FOR i := 1 TO 25 DO
	_Assertions.ThatBool(
		actual := _CollisionDictionary.ContainsKey(key := i),
		message := "Rebuild must preserve dictionary links"
	).IsTrue();
	_Assertions.ThatBool(
		actual := _CollisionSet.Contains(value := i),
		message := "Rebuild must preserve set links"
	).IsTrue();
END_FOR

_CollisionDictionary.Clear();
_CollisionSet.Clear();
_CollisionDictionary.SetCopy(key := _Scalar, value := _OtherScalar);
_CollisionSet.SetCopy(value := _Scalar);
_Assertions.ThatBool(
	actual := _CollisionDictionary.ContainsKey(key := _Scalar),
	message := "Dictionary comparer must survive Clear"
).IsTrue();
_Assertions.ThatBool(
	actual := _CollisionSet.Contains(value := _Scalar),
	message := "Set comparer must survive Clear"
).IsTrue();
END_METHOD

(*!
<summary>Uses matching hashes for cross-width integers, signed zero, NaN and empty descriptors.</summary>
<description>
Starts with independent fixture state. The harness clears persistent resources before publication, including
after an aborted call. Terminal OOM injection is reserved for an isolated test.
</description>
*)
METHOD PRIVATE hashEqualityRepresentations
_Dictionary.SetCopy(key := _SignedKey, value := _Scalar);
_Dictionary.SetCopy(key := _UnsignedKey, value := _OtherScalar);
_Set.SetCopy(value := _SignedKey);
_Set.SetCopy(value := _UnsignedKey);
_Assertions.ThatDInt(
	actual := _Dictionary.Length,
	message := "Equal integer widths must share a key"
).ToBe(expected := 1);
_Assertions.ThatDInt(
	actual := _Set.Length,
	message := "Equal integer widths must share an entry"
).ToBe(expected := 1);

_RealBits.Raw := TOF_Core.Reals.ZERO_BITS;
_Dictionary.SetCopy(key := _RealBits.Value, value := _Scalar);
_Set.SetCopy(value := _RealBits.Value);
_LongRealBits.Raw := NOT TOF_Core.LongReals.MAGNITUDE_MASK;
_Dictionary.SetCopy(key := _LongRealBits.Value, value := _OtherScalar);
_Set.SetCopy(value := _LongRealBits.Value);
_Assertions.ThatDInt(
	actual := _Dictionary.Length,
	message := "Signed floating zeros must share a key"
).ToBe(expected := 2);
_Assertions.ThatDInt(
	actual := _Set.Length,
	message := "Signed floating zeros must share an entry"
).ToBe(expected := 2);

_RealBits.Raw := TOF_Core.Reals.CANONICAL_NAN_BITS;
_LongRealBits.Raw := TOF_Core.LongReals.CANONICAL_NAN_BITS;
_Dictionary.SetCopy(key := _RealBits.Value, value := _Scalar);
_Dictionary.SetCopy(key := _LongRealBits.Value, value := _OtherScalar);
_Set.SetCopy(value := _RealBits.Value);
_Set.SetCopy(value := _LongRealBits.Value);
_Assertions.ThatDInt(
	actual := _Dictionary.Length,
	message := "Cross-width NaNs must share a key"
).ToBe(expected := 3);
_Assertions.ThatDInt(
	actual := _Set.Length,
	message := "Cross-width NaNs must share an entry"
).ToBe(expected := 3);

_Query.Reset();
_Dictionary.SetGeneric(key := _Query, value := _Query);
_Set.SetGeneric(value := _Query);
_Assertions.ThatBool(
	actual := _Dictionary.ContainsGenericKey(key := _Query),
	message := "Empty key must be searchable"
).IsTrue();
_Assertions.ThatBool(
	actual := _Set.ContainsGeneric(value := _Query),
	message := "Empty entry must be searchable"
).IsTrue();
_Assertions.ThatDInt(
	actual := _Dictionary.Length,
	message := "Empty must remain distinct from nonempty values"
).ToBe(expected := 4);
_Assertions.ThatDInt(
	actual := _Set.Length,
	message := "Empty must remain distinct from nonempty values"
).ToBe(expected := 4);
END_METHOD

(*!
<summary>Disposes shared key/value allocations once and retains same-allocation set ownership.</summary>
<description>
Starts with independent fixture state. The harness clears persistent resources before publication, including
after an aborted call. Terminal OOM injection is reserved for an isolated test.
</description>
*)
METHOD PRIVATE hashOwnershipAliases
VAR
	borrowedValue : TOF_Core.GENERIC_VALUE;
	pair : TOF_Core.GENERIC_KEY_VALUE_PAIR;
END_VAR
prepareOwnedValue();
borrowedValue := TOF_Core.GenericValueFactory.FromParts(
	genericTypeClass := _OwnedValue.TypeClass,
	address := _OwnedValue.Address,
	size := _OwnedValue.Size,
	memoryManagementBehavior := TOF_Core.GENERIC_MEMORY_MANAGEMENT_BEHAVIOR.STORE_ORIGINAL_REFERENCE_AND_NOT_OWNS_MEMORY
);
_Dictionary.SetGeneric(key := _OwnedValue, value := _OwnedValue);
_OwnedValue.Reset();
pair := _Dictionary.GetKeyValuePairByIndex(index := 0);
_Assertions.ThatBool(
	actual := pair.Key.IsMemoryOwner,
	message := "Shared pair ownership must belong to key"
).IsTrue();
_Assertions.ThatBool(
	actual := pair.Value.IsMemoryOwner,
	message := "Shared pair value must remain borrowed"
).IsFalse();
_Dictionary.SetGeneric(key := borrowedValue, value := borrowedValue);
_Assertions.ThatUDInt(
	actual := _CloneExitCount,
	message := "Retained pair storage must stay alive"
).ToBe(expected := 0);
_Dictionary.Clear();
_Assertions.ThatUDInt(
	actual := _CloneExitCount,
	message := "Shared pair must be destroyed once"
).ToBe(expected := 1);

prepareOwnedValue();
borrowedValue := TOF_Core.GenericValueFactory.FromParts(
	genericTypeClass := _OwnedValue.TypeClass,
	address := _OwnedValue.Address,
	size := _OwnedValue.Size,
	memoryManagementBehavior := TOF_Core.GENERIC_MEMORY_MANAGEMENT_BEHAVIOR.STORE_ORIGINAL_REFERENCE_AND_NOT_OWNS_MEMORY
);
_Set.SetGeneric(value := _OwnedValue);
_OwnedValue.Reset();
_Set.SetGeneric(value := borrowedValue);
_Assertions.ThatBool(
	actual := _Set.GetByIndex(index := 0).IsMemoryOwner,
	message := "Set replacement must preserve owner"
).IsTrue();
_Set.Clear();
_Assertions.ThatUDInt(
	actual := _CloneExitCount,
	message := "Retained set storage must be destroyed once"
).ToBe(expected := 2);
END_METHOD

(*!
<summary>Preserves ownership when replacing a stored value with its borrowed same-allocation alias.</summary>
<description>
Starts with independent fixture state. The harness clears persistent resources before publication, including
after an aborted call. Terminal OOM injection is reserved for an isolated test.
</description>
*)
METHOD PRIVATE listOwnershipReplacement
VAR
	borrowedValue : TOF_Core.GENERIC_VALUE;
END_VAR
prepareOwnedValue();
_List.AppendGeneric(value := _OwnedValue);
_OwnedValue.Reset();
borrowedValue := TOF_Core.GenericValueFactory.FromParts(
	genericTypeClass := _List.Get(index := 0).TypeClass,
	address := _List.Get(index := 0).Address,
	size := _List.Get(index := 0).Size,
	memoryManagementBehavior := TOF_Core.GENERIC_MEMORY_MANAGEMENT_BEHAVIOR.STORE_ORIGINAL_REFERENCE_AND_NOT_OWNS_MEMORY
);
_List.SetGeneric(index := 0, value := borrowedValue);
_Assertions.ThatBool(
	actual := _List.Get(index := 0).IsMemoryOwner,
	message := "Borrowed replacement must preserve owner"
).IsTrue();
_Assertions.ThatUDInt(
	actual := _CloneExitCount,
	message := "Same allocation must remain alive"
).ToBe(expected := 0);
_List.Clear();
_Assertions.ThatUDInt(
	actual := _CloneExitCount,
	message := "Retained allocation must be destroyed once"
).ToBe(expected := 1);
END_METHOD

(*!
<summary>Applies skip and maxRemoved and preserves completed removals after a predicate failure.</summary>
<description>
Starts with independent fixture state. The harness clears persistent resources before publication, including
after an aborted call. Terminal OOM injection is reserved for an isolated test.
</description>
*)
METHOD PRIVATE listRemovalLimits
VAR
	i : DINT;
	removedCount : DINT;
	rejected : BOOL;
	exceptionCode : __SYSTEM.ExceptionCode;
END_VAR
FOR i := 1 TO 5 DO
	_List.AppendCopy(value := i);
END_FOR

_Predicate.ResetCount();
_List.RemoveMatched(predicate := _Predicate, skip := 1, maxRemoved := 2, removedCount => removedCount);
_Assertions.ThatDInt(
	actual := removedCount,
	message := "Removal must obey the positive limit"
).ToBe(expected := 2);
_Assertions.ThatUDInt(
	actual := _Predicate.CallCount,
	message := "Limit must stop further callbacks"
).ToBe(expected := 3);
_Assertions.ThatDInt(
	actual := _List.Length,
	message := "Two matches must be removed"
).ToBe(expected := 3);
_Assertions.ThatDInt(
	actual := _List.Get(index := 2).AsDInt(),
	message := "Skipped last match must remain"
).ToBe(expected := 5);
_Predicate.ResetCount();
_List.RemoveMatched(predicate := _Predicate, maxRemoved := 0, removedCount => removedCount);
_Assertions.ThatUDInt(
	actual := _Predicate.CallCount,
	message := "Zero limit must not invoke predicate"
).ToBe(expected := 0);
_Assertions.ThatDInt(
	actual := removedCount,
	message := "Zero limit must report no removals"
).ToBe(expected := 0);

_List.Clear();

FOR i := 1 TO 5 DO
	_List.AppendCopy(value := i);
END_FOR

_Predicate.ResetCount();
_Predicate.ThrowOnCall := 2;

__TRY
	_List.RemoveMatched(predicate := _Predicate, removedCount => removedCount);
__CATCH(exceptionCode)
	rejected := TRUE;
	assertOriginalFailure(exceptionCode := exceptionCode, expectedMessage := "Collection predicate rejected");
__ENDTRY

_Assertions.ThatBool(
	actual := rejected,
	message := "Predicate failure must propagate"
).IsTrue();
_Assertions.ThatDInt(
	actual := _List.Length,
	message := "Completed removal must not roll back"
).ToBe(expected := 4);
_Assertions.ThatDInt(
	actual := _List.Get(index := 3).AsDInt(),
	message := "Remaining order must be valid"
).ToBe(expected := 4);
END_METHOD

(*!
<summary>Diagnoses null constructor sources outside FB_init for all six cursors and concrete current views.</summary>
<description>
All six cursors are constructed with null sources without throwing during FB_init. MoveNext, generic
Current and concrete current views must report configuration failure in the current cyclic task. Reset
remains a local cursor operation that does not access the missing source.
</description>
*)
METHOD PRIVATE missingCursorSources
VAR
	i : DINT;
	rejected : BOOL;
	exceptionCode : __SYSTEM.ExceptionCode;
	caughtException : TOF_Core.IException;
	missingException : TOF_Core.IDataMemberNotSpecifiedException;
	currentValue : TOF_Core.GENERIC_VALUE;
	currentByte : BYTE;
	currentPair : TOF_Core.GENERIC_KEY_VALUE_PAIR;
END_VAR
_NullCursors[0] := _NullByteCursor;
_NullCursors[1] := _NullListCursor;
_NullCursors[2] := _NullQueueCursor;
_NullCursors[3] := _NullStackCursor;
_NullCursors[4] := _NullDictionaryCursor;
_NullCursors[5] := _NullSetCursor;

FOR i := 0 TO 5 DO
	rejected := FALSE;

	__TRY
		_NullCursors[i].MoveNext();
	__CATCH(exceptionCode)
		rejected := TRUE;
		caughtException := TOF_Core.ExceptionManager.GetLastException(
			exceptionCode := exceptionCode,
			catchPointNamespaceName := NamespaceName,
			catchPointPOUName := __POUNAME(),
			catchPointPosition := __POSITION()
		);
		_Assertions.ThatBool(
			actual := __QUERYINTERFACE(caughtException, missingException),
			message := "Missing cursor source must report DataMemberNotSpecifiedException"
		).IsTrue();
	__ENDTRY

	_Assertions.ThatBool(
		actual := rejected,
		message := "MoveNext must reject a missing source"
	).IsTrue();
	rejected := FALSE;

	__TRY
		currentValue := _NullCursors[i].Current;
	__CATCH(exceptionCode)
		rejected := TRUE;
		caughtException := TOF_Core.ExceptionManager.GetLastException(
			exceptionCode := exceptionCode,
			catchPointNamespaceName := NamespaceName,
			catchPointPOUName := __POUNAME(),
			catchPointPosition := __POSITION()
		);
		_Assertions.ThatBool(
			actual := __QUERYINTERFACE(caughtException, missingException),
			message := "Missing cursor source must report DataMemberNotSpecifiedException"
		).IsTrue();
	__ENDTRY

	_Assertions.ThatBool(
		actual := rejected,
		message := "Current must reject a missing source"
	).IsTrue();
	_NullCursors[i].Reset();
END_FOR

rejected := FALSE;

__TRY
	currentByte := _NullByteCursor.CurrentByte;
__CATCH(exceptionCode)
	rejected := TRUE;
	caughtException := TOF_Core.ExceptionManager.GetLastException(
		exceptionCode := exceptionCode,
		catchPointNamespaceName := NamespaceName,
		catchPointPOUName := __POUNAME(),
		catchPointPosition := __POSITION()
	);
	_Assertions.ThatBool(
		actual := __QUERYINTERFACE(caughtException, missingException),
		message := "Missing cursor source must report DataMemberNotSpecifiedException"
	).IsTrue();
__ENDTRY

_Assertions.ThatBool(
	actual := rejected,
	message := "Concrete CurrentByte must reject a missing source"
).IsTrue();
rejected := FALSE;

__TRY
	currentPair := _NullDictionaryCursor.CurrentKeyValuePair;
__CATCH(exceptionCode)
	rejected := TRUE;
	caughtException := TOF_Core.ExceptionManager.GetLastException(
		exceptionCode := exceptionCode,
		catchPointNamespaceName := NamespaceName,
		catchPointPOUName := __POUNAME(),
		catchPointPosition := __POSITION()
	);
	_Assertions.ThatBool(
		actual := __QUERYINTERFACE(caughtException, missingException),
		message := "Missing cursor source must report DataMemberNotSpecifiedException"
	).IsTrue();
__ENDTRY

_Assertions.ThatBool(
	actual := rejected,
	message := "Concrete CurrentKeyValuePair must reject a missing source"
).IsTrue();
END_METHOD

(*!
<summary>Retains one clone as a fixture-owned descriptor until acceptance or cleanup.</summary>
*)
METHOD PRIVATE prepareOwnedValue
_OwnedObject := _CloneSource.Clone();
_OwnedValue := TOF_Core.GenericValueFactory.FromParts(
	genericTypeClass := TOF_Core.GENERIC_TYPE_CLASS.OBJECT,
	address := _OwnedObject.SelfAddress,
	size := _OwnedObject.SelfSize,
	memoryManagementBehavior := TOF_Core.GENERIC_MEMORY_MANAGEMENT_BEHAVIOR.STORE_ORIGINAL_REFERENCE_AND_OWNS_MEMORY
);
_OwnedObject := 0;
END_METHOD

(*!
<summary>Prepares persistent resources and raises before the caller can release them.</summary>
*)
METHOD PRIVATE prepareResourcesThenReject
_Enumerator := _List.CreateEnumerator();
prepareOwnedValue();
TOF_Core.Exceptions.ThrowStandard(
	sourceNamespaceName := NamespaceName,
	sourceClassName := ClassName,
	sourcePOUName := __POUNAME(),
	sourcePosition := __POSITION(),
	message := "Collection fixture rejected"
);
END_METHOD

(*!
<summary>Releases owned queries and retains callback diagnostics across cleanup context changes.</summary>
<description>
Starts with independent fixture state. The harness clears persistent resources before publication, including
after an aborted call. Terminal OOM injection is reserved for an isolated test.
</description>
*)
METHOD PRIVATE queryFailureCleanup
VAR
	rejected : BOOL;
	exceptionCode : __SYSTEM.ExceptionCode;
END_VAR
_BorrowedSource := TOF_Core.GenericValueFactory.FromParts(
	genericTypeClass := TOF_Core.GENERIC_TYPE_CLASS.OBJECT,
	address := _CloneSource.SelfAddress,
	size := _CloneSource.SelfSize,
	memoryManagementBehavior := TOF_Core.GENERIC_MEMORY_MANAGEMENT_BEHAVIOR.STORE_ORIGINAL_REFERENCE_AND_NOT_OWNS_MEMORY
);
_List.AppendGeneric(value := _BorrowedSource);
_Queue.EnqueueGeneric(value := _BorrowedSource);
_Stack.PushGeneric(value := _BorrowedSource);
_CollisionDictionary.SetCopy(key := _Scalar, value := _Scalar);
_CollisionSet.SetCopy(value := _Scalar);
_CloneSource.ThrowOnEquality := TRUE;
_Equality.ThrowOnEquality := TRUE;

prepareOwnedValue();
_Query := _OwnedValue;
_OwnedValue.Reset();

rejected := FALSE;
_CloneExitCount := TOF_Core.UnsignedInt32.ZERO;

__TRY
	_List.ContainsGeneric(value := _Query, releaseValue := TRUE);
	_Query.Reset();
__CATCH(exceptionCode)
	_Query.Reset();
	rejected := TRUE;
	assertOriginalFailure(exceptionCode := exceptionCode, expectedMessage := "Collection object equality rejected");
__ENDTRY

_Assertions.ThatBool(
	actual := rejected,
	message := "Failure must propagate"
).IsTrue();
_Assertions.ThatUDInt(
	actual := _CloneExitCount,
	message := "Owned temporary must be released exactly once"
).ToBe(expected := 1);

prepareOwnedValue();
_Query := _OwnedValue;
_OwnedValue.Reset();

rejected := FALSE;
_CloneExitCount := TOF_Core.UnsignedInt32.ZERO;

__TRY
	_Queue.ContainsGeneric(value := _Query, releaseValue := TRUE);
	_Query.Reset();
__CATCH(exceptionCode)
	_Query.Reset();
	rejected := TRUE;
	assertOriginalFailure(exceptionCode := exceptionCode, expectedMessage := "Collection object equality rejected");
__ENDTRY

_Assertions.ThatBool(
	actual := rejected,
	message := "Failure must propagate"
).IsTrue();
_Assertions.ThatUDInt(
	actual := _CloneExitCount,
	message := "Owned temporary must be released exactly once"
).ToBe(expected := 1);

prepareOwnedValue();
_Query := _OwnedValue;
_OwnedValue.Reset();

rejected := FALSE;
_CloneExitCount := TOF_Core.UnsignedInt32.ZERO;

__TRY
	_Stack.ContainsGeneric(value := _Query, releaseValue := TRUE);
	_Query.Reset();
__CATCH(exceptionCode)
	_Query.Reset();
	rejected := TRUE;
	assertOriginalFailure(exceptionCode := exceptionCode, expectedMessage := "Collection object equality rejected");
__ENDTRY

_Assertions.ThatBool(
	actual := rejected,
	message := "Failure must propagate"
).IsTrue();
_Assertions.ThatUDInt(
	actual := _CloneExitCount,
	message := "Owned temporary must be released exactly once"
).ToBe(expected := 1);

prepareOwnedValue();
_Query := _OwnedValue;
_OwnedValue.Reset();

rejected := FALSE;
_CloneExitCount := TOF_Core.UnsignedInt32.ZERO;

__TRY
	_CollisionDictionary.ContainsGenericKey(key := _Query, releaseKey := TRUE);
	_Query.Reset();
__CATCH(exceptionCode)
	_Query.Reset();
	rejected := TRUE;
	assertOriginalFailure(exceptionCode := exceptionCode, expectedMessage := "Collection equality rejected");
__ENDTRY

_Assertions.ThatBool(
	actual := rejected,
	message := "Failure must propagate"
).IsTrue();
_Assertions.ThatUDInt(
	actual := _CloneExitCount,
	message := "Owned temporary must be released exactly once"
).ToBe(expected := 1);

prepareOwnedValue();
_Query := _OwnedValue;
_OwnedValue.Reset();

rejected := FALSE;
_CloneExitCount := TOF_Core.UnsignedInt32.ZERO;

__TRY
	_CollisionDictionary.GetGenericKeyPosition(key := _Query, releaseKey := TRUE);
	_Query.Reset();
__CATCH(exceptionCode)
	_Query.Reset();
	rejected := TRUE;
	assertOriginalFailure(exceptionCode := exceptionCode, expectedMessage := "Collection equality rejected");
__ENDTRY

_Assertions.ThatBool(
	actual := rejected,
	message := "Failure must propagate"
).IsTrue();
_Assertions.ThatUDInt(
	actual := _CloneExitCount,
	message := "Owned temporary must be released exactly once"
).ToBe(expected := 1);

prepareOwnedValue();
_Query := _OwnedValue;
_OwnedValue.Reset();

rejected := FALSE;
_CloneExitCount := TOF_Core.UnsignedInt32.ZERO;

__TRY
	_CollisionSet.ContainsGeneric(value := _Query, releaseValue := TRUE);
	_Query.Reset();
__CATCH(exceptionCode)
	_Query.Reset();
	rejected := TRUE;
	assertOriginalFailure(exceptionCode := exceptionCode, expectedMessage := "Collection equality rejected");
__ENDTRY

_Assertions.ThatBool(
	actual := rejected,
	message := "Failure must propagate"
).IsTrue();
_Assertions.ThatUDInt(
	actual := _CloneExitCount,
	message := "Owned temporary must be released exactly once"
).ToBe(expected := 1);

prepareOwnedValue();
_Query := _OwnedValue;
_OwnedValue.Reset();

rejected := FALSE;
_CloneExitCount := TOF_Core.UnsignedInt32.ZERO;

__TRY
	_CollisionSet.GetGenericValuePosition(value := _Query, releaseValue := TRUE);
	_Query.Reset();
__CATCH(exceptionCode)
	_Query.Reset();
	rejected := TRUE;
	assertOriginalFailure(exceptionCode := exceptionCode, expectedMessage := "Collection equality rejected");
__ENDTRY

_Assertions.ThatBool(
	actual := rejected,
	message := "Failure must propagate"
).IsTrue();
_Assertions.ThatUDInt(
	actual := _CloneExitCount,
	message := "Owned temporary must be released exactly once"
).ToBe(expected := 1);

_Assertions.ThatDInt(
	actual := _List.Length,
	message := "Failed query must not remove list entries"
).ToBe(expected := 1);
_Assertions.ThatDInt(
	actual := _CollisionDictionary.Length,
	message := "Failed query must not mutate keys"
).ToBe(expected := 1);
_Assertions.ThatDInt(
	actual := _CollisionSet.Length,
	message := "Failed query must not mutate values"
).ToBe(expected := 1);
END_METHOD

(*!
<summary>Invokes the validator once per enqueue and rejects before growth or adoption.</summary>
<description>
Starts with independent fixture state. The harness clears persistent resources before publication, including
after an aborted call. Terminal OOM injection is reserved for an isolated test.
</description>
*)
METHOD PRIVATE queueValidationAndGrowth
VAR
	i : DINT;
	rejected : BOOL;
	exceptionCode : __SYSTEM.ExceptionCode;
END_VAR
_Queue.DefaultDynamicAllocationElementCount := 2;
_Validator.ResetCount();

FOR i := 1 TO 6 DO
	_Queue.EnqueueCopy(value := i);
END_FOR

_Assertions.ThatUDInt(
	actual := _Validator.CallCount,
	message := "Enqueue must validate exactly once"
).ToBe(expected := 6);
_Assertions.ThatDInt(
	actual := _Queue.Capacity,
	message := "Queue must grow several times"
).ToBe(expected := 6);
_Validator.Reject := TRUE;
prepareOwnedValue();

__TRY
	_Queue.EnqueueGeneric(value := _OwnedValue);
__CATCH(exceptionCode)
	rejected := TRUE;
	assertOriginalFailure(exceptionCode := exceptionCode, expectedMessage := "Collection validation rejected");
__ENDTRY

_Assertions.ThatBool(
	actual := rejected,
	message := "Configured validator must reject"
).IsTrue();
_Assertions.ThatDInt(
	actual := _Queue.Capacity,
	message := "Rejected enqueue must not grow"
).ToBe(expected := 6);
_Assertions.ThatDInt(
	actual := _Queue.Length,
	message := "Rejected enqueue must not insert"
).ToBe(expected := 6);
_Assertions.ThatUDInt(
	actual := _CloneExitCount,
	message := "Rejected owner must remain caller-owned"
).ToBe(expected := 0);
_OwnedValue.Release();
_Assertions.ThatUDInt(
	actual := _CloneExitCount,
	message := "Caller must retain disposal rights"
).ToBe(expected := 1);
_Validator.Reject := FALSE;

FOR i := 1 TO 6 DO
	_Assertions.ThatDInt(
		actual := _Queue.Peek().AsDInt(),
		message := "Growth must preserve FIFO order"
	).ToBe(expected := i);
	_Queue.RemoveFirst();
END_FOR
END_METHOD

(*!
<summary>Releases persistent cursor ownership without deleting source collections.</summary>
<description>
Clears interface aliases before best-effort disposal. Latches failed disposal or duplicate ownership.
</description>
*)
METHOD PRIVATE releaseCursors
VAR
	ownedCursor : TOF_Core.IObject;
END_VAR
IF _Enumerator <> 0 AND_THEN _Enumerator = _SecondEnumerator THEN
	_SecondEnumerator := 0;
	_ReleaseFailed := TRUE;
END_IF

IF _Enumerator <> 0 THEN
	ownedCursor := _Enumerator;
	_Enumerator := 0;

	IF NOT TOF_Core.Memory.TryReleaseDynamicObject(instance := ownedCursor) THEN
		_ReleaseFailed := TRUE;
	END_IF
END_IF

IF _SecondEnumerator <> 0 THEN
	ownedCursor := _SecondEnumerator;
	_SecondEnumerator := 0;

	IF NOT TOF_Core.Memory.TryReleaseDynamicObject(instance := ownedCursor) THEN
		_ReleaseFailed := TRUE;
	END_IF
END_IF
END_METHOD

(*!
<summary>Releases the prepared dictionary key if the second object clone rejects.</summary>
<description>
Starts with independent fixture state. The harness clears persistent resources before publication, including
after an aborted call. Terminal OOM injection is reserved for an isolated test.
</description>
*)
METHOD PRIVATE secondCopyFailureCleanup
VAR
	rejected : BOOL;
	exceptionCode : __SYSTEM.ExceptionCode;
END_VAR
_FailingCloneSource.ThrowOnClone := TRUE;

rejected := FALSE;
_CloneExitCount := TOF_Core.UnsignedInt32.ZERO;

__TRY
	_Dictionary.SetCopy(
		key := _CloneSource,
		value := _FailingCloneSource,
		keyIsObject := TRUE,
		valueIsObject := TRUE
	);
__CATCH(exceptionCode)
	rejected := TRUE;
	assertOriginalFailure(exceptionCode := exceptionCode, expectedMessage := "Collection clone rejected");
__ENDTRY

_Assertions.ThatBool(
	actual := rejected,
	message := "Failure must propagate"
).IsTrue();
_Assertions.ThatUDInt(
	actual := _CloneExitCount,
	message := "Owned temporary must be released exactly once"
).ToBe(expected := 1);

_Assertions.ThatBool(
	actual := _Dictionary.Empty,
	message := "Second clone failure must not insert a pair"
).IsTrue();
END_METHOD

(*!
<summary>Retains every owned descriptor after comparer failures in both sorting branches.</summary>
<description>
Starts with independent fixture state. The harness clears persistent resources before publication, including
after an aborted call. Terminal OOM injection is reserved for an isolated test.
</description>
*)
METHOD PRIVATE sortFailurePreservesEntries
VAR
	i : DINT;
	count : DINT;
	rejected : BOOL;
	exceptionCode : __SYSTEM.ExceptionCode;
END_VAR
FOR count := 16 TO 17 DO
	_List.Clear();

	FOR i := count TO 1 BY -1 DO
		_List.AppendCopy(value := i);
	END_FOR

	_Comparer.ResetCount();
	_Comparer.ThrowOnCall := 3;
	rejected := FALSE;

	__TRY
		_List.Sort(comparer := _Comparer);
	__CATCH(exceptionCode)
		rejected := TRUE;
		assertOriginalFailure(exceptionCode := exceptionCode, expectedMessage := "Collection comparer rejected");
	__ENDTRY

	_Assertions.ThatBool(
		actual := rejected,
		message := "Comparer failure must propagate"
	).IsTrue();
	_Assertions.ThatDInt(
		actual := _List.Length,
		message := "Failed sort must preserve Length"
	).ToBe(expected := count);
	_Comparer.ThrowOnCall := 0;
	_List.Sort(comparer := _Comparer);

	FOR i := 0 TO count - 1 DO
		_Assertions.ThatDInt(
			actual := _List.Get(index := i).AsDInt(),
			message := "Failed sorting must neither lose nor duplicate entries"
		).ToBe(expected := i + 1);
		_Assertions.ThatBool(
			actual := _List.Get(index := i).IsMemoryOwner,
			message := "Sorting must preserve ownership"
		).IsTrue();
	END_FOR
END_FOR
END_METHOD

(*!
<summary>Retains static-full diagnostics and disposes prepared copies before adoption.</summary>
<description>
Starts with independent fixture state. The harness clears persistent resources before publication, including
after an aborted call. Terminal OOM injection is reserved for an isolated test.
</description>
*)
METHOD PRIVATE staticFullCopyCleanup
VAR
	rejected : BOOL;
	exceptionCode : __SYSTEM.ExceptionCode;
	caughtException : TOF_Core.IException;
	fullException : TOF_Core.IStaticCollectionFullException;
END_VAR
_FullList.AppendCopy(value := _Scalar);
_FullQueue.EnqueueCopy(value := _Scalar);
_FullStack.PushCopy(value := _Scalar);
_FullDictionary.SetCopy(key := _Scalar, value := _Scalar);
_FullSet.SetCopy(value := _Scalar);

rejected := FALSE;
_CloneExitCount := TOF_Core.UnsignedInt32.ZERO;

__TRY
	_FullList.AppendCopy(value := _CloneSource, isObject := TRUE);
__CATCH(exceptionCode)
	rejected := TRUE;
	caughtException := TOF_Core.ExceptionManager.GetLastException(
		exceptionCode := exceptionCode,
		catchPointNamespaceName := NamespaceName,
		catchPointPOUName := __POUNAME(),
		catchPointPosition := __POSITION()
	);
	_Assertions.ThatBool(
		actual := __QUERYINTERFACE(caughtException, fullException),
		message := "Static-full diagnostic must survive clone disposal"
	).IsTrue();
__ENDTRY

_Assertions.ThatBool(
	actual := rejected,
	message := "Static full must reject Copy"
).IsTrue();
_Assertions.ThatUDInt(
	actual := _CloneExitCount,
	message := "Rejected copy must be released once"
).ToBe(expected := 1);

rejected := FALSE;
_CloneExitCount := TOF_Core.UnsignedInt32.ZERO;

__TRY
	_FullList.InsertCopy(index := 0, value := _CloneSource, isObject := TRUE);
__CATCH(exceptionCode)
	rejected := TRUE;
	caughtException := TOF_Core.ExceptionManager.GetLastException(
		exceptionCode := exceptionCode,
		catchPointNamespaceName := NamespaceName,
		catchPointPOUName := __POUNAME(),
		catchPointPosition := __POSITION()
	);
	_Assertions.ThatBool(
		actual := __QUERYINTERFACE(caughtException, fullException),
		message := "Static-full diagnostic must survive clone disposal"
	).IsTrue();
__ENDTRY

_Assertions.ThatBool(
	actual := rejected,
	message := "Static full must reject Copy"
).IsTrue();
_Assertions.ThatUDInt(
	actual := _CloneExitCount,
	message := "Rejected copy must be released once"
).ToBe(expected := 1);

rejected := FALSE;
_CloneExitCount := TOF_Core.UnsignedInt32.ZERO;

__TRY
	_FullQueue.EnqueueCopy(value := _CloneSource, isObject := TRUE);
__CATCH(exceptionCode)
	rejected := TRUE;
	caughtException := TOF_Core.ExceptionManager.GetLastException(
		exceptionCode := exceptionCode,
		catchPointNamespaceName := NamespaceName,
		catchPointPOUName := __POUNAME(),
		catchPointPosition := __POSITION()
	);
	_Assertions.ThatBool(
		actual := __QUERYINTERFACE(caughtException, fullException),
		message := "Static-full diagnostic must survive clone disposal"
	).IsTrue();
__ENDTRY

_Assertions.ThatBool(
	actual := rejected,
	message := "Static full must reject Copy"
).IsTrue();
_Assertions.ThatUDInt(
	actual := _CloneExitCount,
	message := "Rejected copy must be released once"
).ToBe(expected := 1);

rejected := FALSE;
_CloneExitCount := TOF_Core.UnsignedInt32.ZERO;

__TRY
	_FullStack.PushCopy(value := _CloneSource, isObject := TRUE);
__CATCH(exceptionCode)
	rejected := TRUE;
	caughtException := TOF_Core.ExceptionManager.GetLastException(
		exceptionCode := exceptionCode,
		catchPointNamespaceName := NamespaceName,
		catchPointPOUName := __POUNAME(),
		catchPointPosition := __POSITION()
	);
	_Assertions.ThatBool(
		actual := __QUERYINTERFACE(caughtException, fullException),
		message := "Static-full diagnostic must survive clone disposal"
	).IsTrue();
__ENDTRY

_Assertions.ThatBool(
	actual := rejected,
	message := "Static full must reject Copy"
).IsTrue();
_Assertions.ThatUDInt(
	actual := _CloneExitCount,
	message := "Rejected copy must be released once"
).ToBe(expected := 1);

rejected := FALSE;
_CloneExitCount := TOF_Core.UnsignedInt32.ZERO;

__TRY
	_FullDictionary.SetCopy(key := _OtherScalar, value := _CloneSource, valueIsObject := TRUE);
__CATCH(exceptionCode)
	rejected := TRUE;
	caughtException := TOF_Core.ExceptionManager.GetLastException(
		exceptionCode := exceptionCode,
		catchPointNamespaceName := NamespaceName,
		catchPointPOUName := __POUNAME(),
		catchPointPosition := __POSITION()
	);
	_Assertions.ThatBool(
		actual := __QUERYINTERFACE(caughtException, fullException),
		message := "Static-full diagnostic must survive clone disposal"
	).IsTrue();
__ENDTRY

_Assertions.ThatBool(
	actual := rejected,
	message := "Static full must reject Copy"
).IsTrue();
_Assertions.ThatUDInt(
	actual := _CloneExitCount,
	message := "Rejected copy must be released once"
).ToBe(expected := 1);

rejected := FALSE;
_CloneExitCount := TOF_Core.UnsignedInt32.ZERO;

__TRY
	_FullSet.SetCopy(value := _CloneSource, isObject := TRUE);
__CATCH(exceptionCode)
	rejected := TRUE;
	caughtException := TOF_Core.ExceptionManager.GetLastException(
		exceptionCode := exceptionCode,
		catchPointNamespaceName := NamespaceName,
		catchPointPOUName := __POUNAME(),
		catchPointPosition := __POSITION()
	);
	_Assertions.ThatBool(
		actual := __QUERYINTERFACE(caughtException, fullException),
		message := "Static-full diagnostic must survive clone disposal"
	).IsTrue();
__ENDTRY

_Assertions.ThatBool(
	actual := rejected,
	message := "Static full must reject Copy"
).IsTrue();
_Assertions.ThatUDInt(
	actual := _CloneExitCount,
	message := "Rejected copy must be released once"
).ToBe(expected := 1);

_Assertions.ThatDInt(
	actual := _FullList.Length,
	message := "Full list must retain its entry"
).ToBe(expected := 1);
_Assertions.ThatDInt(
	actual := _FullQueue.Length,
	message := "Full queue must retain its entry"
).ToBe(expected := 1);
_Assertions.ThatDInt(
	actual := _FullStack.Length,
	message := "Full stack must retain its entry"
).ToBe(expected := 1);
_Assertions.ThatDInt(
	actual := _FullDictionary.Length,
	message := "Full dictionary must retain its entry"
).ToBe(expected := 1);
_Assertions.ThatDInt(
	actual := _FullSet.Length,
	message := "Full set must retain its entry"
).ToBe(expected := 1);
END_METHOD

(*!
<summary>Contains hash and equality failures in all six Try methods and still releases owned queries.</summary>
<description>
Starts with independent fixture state. The harness clears persistent resources before publication, including
after an aborted call. Terminal OOM injection is reserved for an isolated test.
</description>
*)
METHOD PRIVATE containsCollectionCallbackFailures
VAR
	failureKind : DINT;
	found : BOOL;
	escaped : BOOL;
	foundValue : TOF_Core.GENERIC_VALUE;
END_VAR
_CollisionDictionary.SetCopy(key := _Scalar, value := _Scalar);
_CollisionSet.SetCopy(value := _Scalar);

FOR failureKind := 0 TO 1 DO
	_Equality.ThrowOnHash := failureKind = 0;
	_Equality.ThrowOnEquality := failureKind = 1;

	found := TRUE;
	escaped := FALSE;

	__TRY
		found := _CollisionDictionary.TryGetValueByKey(key := _OtherScalar, value => foundValue);
	__CATCH
		escaped := TRUE;
	__ENDTRY

	_Assertions.ThatBool(
		actual := escaped,
		message := "Try callback failure must not escape"
	).IsFalse();
	_Assertions.ThatBool(
		actual := found,
		message := "Try callback failure must report failure"
	).IsFalse();

	prepareOwnedValue();
	_Query := _OwnedValue;
	_OwnedValue.Reset();
	_CloneExitCount := TOF_Core.UnsignedInt32.ZERO;
	found := TRUE;
	escaped := FALSE;

	__TRY
		found := _CollisionDictionary.TryGetValueByGenericKey(key := _Query, releaseKey := TRUE, value => foundValue);
	__CATCH
		escaped := TRUE;
	__ENDTRY

	_Assertions.ThatBool(
		actual := escaped,
		message := "Try callback failure must not escape"
	).IsFalse();
	_Assertions.ThatBool(
		actual := found,
		message := "Try callback failure must report failure"
	).IsFalse();
	_Query.Reset();
	_Assertions.ThatUDInt(
		actual := _CloneExitCount,
		message := "Failed Try must dispose its owned query"
	).ToBe(expected := 1);

	found := TRUE;
	escaped := FALSE;

	__TRY
		_CollisionDictionary.TryRemoveByKey(key := _OtherScalar, removed => found);
	__CATCH
		escaped := TRUE;
	__ENDTRY

	_Assertions.ThatBool(
		actual := escaped,
		message := "Try callback failure must not escape"
	).IsFalse();
	_Assertions.ThatBool(
		actual := found,
		message := "Try callback failure must report failure"
	).IsFalse();

	prepareOwnedValue();
	_Query := _OwnedValue;
	_OwnedValue.Reset();
	_CloneExitCount := TOF_Core.UnsignedInt32.ZERO;
	found := TRUE;
	escaped := FALSE;

	__TRY
		_CollisionDictionary.TryRemoveByGenericKey(key := _Query, releaseKey := TRUE, removed => found);
	__CATCH
		escaped := TRUE;
	__ENDTRY

	_Assertions.ThatBool(
		actual := escaped,
		message := "Try callback failure must not escape"
	).IsFalse();
	_Assertions.ThatBool(
		actual := found,
		message := "Try callback failure must report failure"
	).IsFalse();
	_Query.Reset();
	_Assertions.ThatUDInt(
		actual := _CloneExitCount,
		message := "Failed Try must dispose its owned query"
	).ToBe(expected := 1);

	found := TRUE;
	escaped := FALSE;

	__TRY
		_CollisionSet.TryRemove(value := _OtherScalar, removed => found);
	__CATCH
		escaped := TRUE;
	__ENDTRY

	_Assertions.ThatBool(
		actual := escaped,
		message := "Try callback failure must not escape"
	).IsFalse();
	_Assertions.ThatBool(
		actual := found,
		message := "Try callback failure must report failure"
	).IsFalse();

	prepareOwnedValue();
	_Query := _OwnedValue;
	_OwnedValue.Reset();
	_CloneExitCount := TOF_Core.UnsignedInt32.ZERO;
	found := TRUE;
	escaped := FALSE;

	__TRY
		_CollisionSet.TryRemoveGeneric(value := _Query, releaseValue := TRUE, removed => found);
	__CATCH
		escaped := TRUE;
	__ENDTRY

	_Assertions.ThatBool(
		actual := escaped,
		message := "Try callback failure must not escape"
	).IsFalse();
	_Assertions.ThatBool(
		actual := found,
		message := "Try callback failure must report failure"
	).IsFalse();
	_Query.Reset();
	_Assertions.ThatUDInt(
		actual := _CloneExitCount,
		message := "Failed Try must dispose its owned query"
	).ToBe(expected := 1);
END_FOR

_Assertions.ThatDInt(
	actual := _CollisionDictionary.Length,
	message := "Failed Try must preserve dictionary"
).ToBe(expected := 1);
_Assertions.ThatDInt(
	actual := _CollisionSet.Length,
	message := "Failed Try must preserve set"
).ToBe(expected := 1);
_Assertions.ThatBool(
	actual := TOF_Core.DynamicMemoryManager.HasAllocationFailed,
	message := "Ordinary rejection is not OOM"
).IsFalse();
END_METHOD

(*!
<summary>Borrows the concrete fixture class name.</summary>
*)
{attribute 'monitoring' := 'call'}
PROPERTY ClassName : REFERENCE TO STRING
GET
ClassName REF= _ClassName;
END_GET
END_PROPERTY

(*!
<summary>Borrows the test namespace for diagnostic context.</summary>
*)
{attribute 'monitoring' := 'call'}
PROPERTY NamespaceName : REFERENCE TO STRING
GET
NamespaceName REF= CurrentNamespace.Name;
END_GET
END_PROPERTY

(*!
<summary>Reports the complete fixture instance size, excluding separately allocated storage.</summary>
*)
{attribute 'monitoring' := 'call'}
PROPERTY SelfSize : ULINT
GET
SelfSize := XSIZEOF(THIS^);
END_GET
END_PROPERTY

END_FUNCTION_BLOCK

// ---- Tests/Collections/Contract/CollectionComparableProbe.TcPOU
(*
SPDX-FileCopyrightText: © 2026 Oleksandr Tiutyk <trofimich@gmail.com>
SPDX-License-Identifier: MIT
License: https://opensource.org/license/mit
*)

(*!
<summary>Provides a scalar natural order for borrowed OBJECT list entries.</summary>
<description>
Supports other ICollectionSortValue objects. Comparisons copy the other scalar key without mutating or
retaining either object. The caller keeps sort keys stable during sorting; no allocation or cleanup is used.
</description>
*)

FUNCTION_BLOCK CollectionComparableProbe EXTENDS TOF_Core.Object IMPLEMENTS ICollectionSortValue
VAR_INPUT
	//! <summary>Scalar key defining the fixture's natural order.</summary>
	SortValue : DINT;
END_VAR
VAR_STAT
	_ClassName : STRING := __POUNAME();
END_VAR

(*!
<summary>Provides the concrete test fixture class name.</summary>
*)
{attribute 'monitoring' := 'call'}
PROPERTY ClassName : REFERENCE TO STRING
GET
ClassName REF= _ClassName;
END_GET
END_PROPERTY

(*!
<summary>Compares supported scalar-key objects and rejects null or unrelated comparable types.</summary>
*)
METHOD CompareTo : TOF_Core.COMPARISON_RESULT
VAR_IN_OUT CONSTANT
	otherValue : TOF_Core.IComparable;
END_VAR
VAR
	otherSortValue : ICollectionSortValue;
	otherKey : DINT;
END_VAR
IF otherValue = 0 THEN
	TOF_Core.Exceptions.ThrowArgumentNotSpecified(
		sourceNamespaceName := NamespaceName,
		sourceClassName := ClassName,
		sourcePOUName := __POUNAME(),
		sourcePosition := __POSITION(),
		argumentName := 'otherValue'
	);
END_IF

IF NOT __QUERYINTERFACE(otherValue, otherSortValue) THEN
	TOF_Core.Exceptions.ThrowStandard(
		sourceNamespaceName := NamespaceName,
		sourceClassName := ClassName,
		sourcePOUName := __POUNAME(),
		sourcePosition := __POSITION(),
		message := "Unsupported collection comparable fixture"
	);
END_IF

otherKey := otherSortValue.GetSortValue();

IF SortValue < otherKey THEN
	CompareTo := TOF_Core.COMPARISON_RESULT.FIRST_LESS_THAN_SECOND;
ELSIF SortValue > otherKey THEN
	CompareTo := TOF_Core.COMPARISON_RESULT.FIRST_GREATER_THAN_SECOND;
ELSE
	CompareTo := TOF_Core.COMPARISON_RESULT.FIRST_EQUAL_TO_SECOND;
END_IF
END_METHOD

(*!
<summary>Copies the configured sort key without mutation.</summary>
*)
METHOD GetSortValue : DINT
GetSortValue := SortValue;
END_METHOD

(*!
<summary>Borrows the compiler-initialized test namespace.</summary>
*)
{attribute 'monitoring' := 'call'}
PROPERTY NamespaceName : REFERENCE TO STRING
GET
NamespaceName REF= CurrentNamespace.Name;
END_GET
END_PROPERTY

(*!
<summary>Reports the complete fixture instance size, excluding separately allocated storage.</summary>
*)
{attribute 'monitoring' := 'call'}
PROPERTY SelfSize : ULINT
GET
SelfSize := XSIZEOF(THIS^);
END_GET
END_PROPERTY

END_FUNCTION_BLOCK

// ---- Tests/Collections/Contract/CollectionCloneProbe.TcPOU
(*
SPDX-FileCopyrightText: © 2026 Oleksandr Tiutyk <trofimich@gmail.com>
SPDX-License-Identifier: MIT
License: https://opensource.org/license/mit
*)

(*!
<summary>Creates caller-owned clones that observe disposal and can invalidate exception transport.</summary>
<description>
The source is persistent. Clones borrow a persistent counter and belong exclusively to their recipient.
Clone can reject before allocation. A selected clone clears only the current task's borrowed exception slot
on disposal, modelling cleanup context changes without throwing, allocating or registering exceptions in
FB_exit. The source itself never clears transport. Do not copy source or clone instances by value.
No cross-task access is supported.
</description>
*)

{attribute 'enable_dynamic_creation'}
FUNCTION_BLOCK CollectionCloneProbe EXTENDS TOF_Core.Object IMPLEMENTS TOF_Core.ICloneable
VAR_INPUT
	//! <summary>Rejects default object equality callbacks without changing either operand.</summary>
	ThrowOnEquality : BOOL;
	//! <summary>Rejects Clone before allocating a result.</summary>
	ThrowOnClone : BOOL;
	//! <summary>Makes subsequent clones drop the current task's borrowed exception slot during disposal.</summary>
	ClearCloneTransportOnExit : BOOL;
END_VAR
VAR_STAT
	_ClassName : STRING := __POUNAME();
END_VAR
VAR
	_ExitCounter : REFERENCE TO UDINT;
	_ClearTransportOnExit : BOOL;
END_VAR

(*!
<summary>Provides the concrete test fixture class name.</summary>
*)
{attribute 'monitoring' := 'call'}
PROPERTY ClassName : REFERENCE TO STRING
GET
ClassName REF= _ClassName;
END_GET
END_PROPERTY

(*!
<summary>Creates one independently owned probe or raises before returning.</summary>
<description>
Does not register its result for automatic cleanup. The caller owns it and must release or transfer it.
The source's counter is borrowed; failure before NEW leaves source and counter unchanged.
</description>
*)
METHOD Clone : TOF_Core.IObject
VAR
	clonePointer : POINTER TO CollectionCloneProbe;
END_VAR
IF ThrowOnClone THEN
	TOF_Core.Exceptions.ThrowStandard(
		sourceNamespaceName := NamespaceName,
		sourceClassName := ClassName,
		sourcePOUName := __POUNAME(),
		sourcePosition := __POSITION(),
		message := "Collection clone rejected"
	);
END_IF

clonePointer := __NEW(CollectionCloneProbe);

IF clonePointer = 0 THEN
	TOF_Core.DynamicMemoryManager.RaiseAllocationFailure();
END_IF

IF __ISVALIDREF(_ExitCounter) THEN
	clonePointer^._ExitCounter REF= _ExitCounter;
END_IF
clonePointer^._ClearTransportOnExit := ClearCloneTransportOnExit;
Clone := clonePointer^;
END_METHOD

(*!
<summary>Uses identity equality or raises the configured callback failure.</summary>
<description>
Does not mutate or retain the compared object. Default identity hashes remain consistent when not rejecting.
</description>
*)
METHOD Equals : BOOL
VAR_INPUT
	other : TOF_Core.IObject;
END_VAR
IF ThrowOnEquality THEN
	TOF_Core.Exceptions.ThrowStandard(
		sourceNamespaceName := NamespaceName,
		sourceClassName := ClassName,
		sourcePOUName := __POUNAME(),
		sourcePosition := __POSITION(),
		message := "Collection object equality rejected"
	);
END_IF

Equals := SUPER^.Equals(other := other);
END_METHOD

(*!
<summary>Observes destruction and optionally drops current-task exception transport.</summary>
<description>
Does not raise, allocate or register exceptions. Guards the cyclic task context before touching transport;
the borrowed counter is persistent. Dropping transport does not free registered exception payloads.
</description>
*)
METHOD FB_exit : BOOL
VAR_INPUT
	bInCopyCode : BOOL;
END_VAR
VAR
	taskIndex : DINT;
END_VAR
IF __ISVALIDREF(_ExitCounter) THEN
	_ExitCounter := _ExitCounter + 1;
END_IF

IF _ClearTransportOnExit THEN
	taskIndex := TOF_Core.System.GetCurrentTaskIndex();

	IF taskIndex > TOF_Core.SignedInt32.ZERO AND_THEN taskIndex <= TOF_Core.System.TASK_COUNT THEN
		TOF_Core.ExceptionManager.Cleanup();
	END_IF
END_IF
END_METHOD

(*!
<summary>Borrows the compiler-initialized test namespace.</summary>
*)
{attribute 'monitoring' := 'call'}
PROPERTY NamespaceName : REFERENCE TO STRING
GET
NamespaceName REF= CurrentNamespace.Name;
END_GET
END_PROPERTY

(*!
<summary>Binds the persistent counter borrowed by subsequent clones.</summary>
<description>
The counter must remain alive until every clone and the source have been destroyed.
</description>
*)
METHOD ObserveExit
VAR_IN_OUT
	counter : UDINT;
END_VAR
_ExitCounter REF= counter;
END_METHOD

(*!
<summary>Reports the complete fixture instance size, excluding separately allocated storage.</summary>
*)
{attribute 'monitoring' := 'call'}
PROPERTY SelfSize : ULINT
GET
SelfSize := XSIZEOF(THIS^);
END_GET
END_PROPERTY

END_FUNCTION_BLOCK

// ---- Tests/Collections/Contract/CollectionValidatorProbe.TcPOU
(*
SPDX-FileCopyrightText: © 2026 Oleksandr Tiutyk <trofimich@gmail.com>
SPDX-License-Identifier: MIT
License: https://opensource.org/license/mit
*)

(*!
<summary>Counts validation calls and optionally rejects a borrowed descriptor.</summary>
<description>
Used by persistent collection fixtures. Rejection changes only the call counter and propagates StandardException.
</description>
*)

FUNCTION_BLOCK CollectionValidatorProbe EXTENDS TOF_Core.Object IMPLEMENTS TOF_Core.IGenericValueValidator
VAR_INPUT
	//! <summary>Rejects every value after counting the call.</summary>
	Reject : BOOL;
END_VAR
VAR_OUTPUT
	//! <summary>Number of completed entries to Validate since ResetCount.</summary>
	CallCount : UDINT;
END_VAR
VAR_STAT
	_ClassName : STRING := __POUNAME();
END_VAR

(*!
<summary>Provides the concrete test fixture class name.</summary>
*)
{attribute 'monitoring' := 'call'}
PROPERTY ClassName : REFERENCE TO STRING
GET
ClassName REF= _ClassName;
END_GET
END_PROPERTY

(*!
<summary>Borrows the compiler-initialized test namespace.</summary>
*)
{attribute 'monitoring' := 'call'}
PROPERTY NamespaceName : REFERENCE TO STRING
GET
NamespaceName REF= CurrentNamespace.Name;
END_GET
END_PROPERTY

(*!
<summary>Resets only the observed validation call count.</summary>
*)
METHOD ResetCount
CallCount := TOF_Core.UnsignedInt32.ZERO;
END_METHOD

(*!
<summary>Reports the complete fixture instance size, excluding separately allocated storage.</summary>
*)
{attribute 'monitoring' := 'call'}
PROPERTY SelfSize : ULINT
GET
SelfSize := XSIZEOF(THIS^);
END_GET
END_PROPERTY

(*!
<summary>Counts the call and rejects when configured without adopting the descriptor.</summary>
*)
METHOD Validate
VAR_INPUT
	validatedObjectName : WSTRING;
END_VAR
VAR_IN_OUT CONSTANT
	valueToValidate : TOF_Core.GENERIC_VALUE;
END_VAR
CallCount := CallCount + 1;

IF Reject THEN
	TOF_Core.Exceptions.ThrowStandard(
		sourceNamespaceName := NamespaceName,
		sourceClassName := ClassName,
		sourcePOUName := __POUNAME(),
		sourcePosition := __POSITION(),
		message := "Collection validation rejected"
	);
END_IF
END_METHOD

END_FUNCTION_BLOCK

// ---- Tests/Collections/Contract/CollectionEqualityProbe.TcPOU
(*
SPDX-FileCopyrightText: © 2026 Oleksandr Tiutyk <trofimich@gmail.com>
SPDX-License-Identifier: MIT
License: https://opensource.org/license/mit
*)

(*!
<summary>Provides default value equality with controlled collisions and callback failures.</summary>
<description>
Constant hash codes deliberately exercise chains. Equality delegates to GENERIC_VALUE defaults without
recursively supplying this strategy. MatchEveryValue selects a universal equivalence relation with the same
constant hash. Its value stays fixed while entries are stored. Failure-injection flags do not change
successful equality or hash results.
</description>
*)

FUNCTION_BLOCK CollectionEqualityProbe EXTENDS TOF_Core.Object IMPLEMENTS TOF_Core.IEqualityComparer
VAR_INPUT
	//! <summary>Selects universal equality before populating a query-matrix container.</summary>
	MatchEveryValue : BOOL;
	//! <summary>Rejects the next and subsequent hash callbacks until cleared.</summary>
	ThrowOnHash : BOOL;
	//! <summary>Rejects equality callbacks until cleared.</summary>
	ThrowOnEquality : BOOL;
END_VAR
VAR_STAT
	_ClassName : STRING := __POUNAME();
END_VAR

(*!
<summary>Compares borrowed descriptors or raises the configured equality failure.</summary>
*)
METHOD AreEqual : BOOL
VAR_INPUT
	first : TOF_Core.GENERIC_VALUE;
	second : TOF_Core.GENERIC_VALUE;
END_VAR
IF ThrowOnEquality THEN
	TOF_Core.Exceptions.ThrowStandard(
		sourceNamespaceName := NamespaceName,
		sourceClassName := ClassName,
		sourcePOUName := __POUNAME(),
		sourcePosition := __POSITION(),
		message := "Collection equality rejected"
	);
END_IF

IF MatchEveryValue THEN
	AreEqual := TRUE;
ELSE
	AreEqual := first.Equals(otherValue := second);
END_IF
END_METHOD

(*!
<summary>Provides the concrete test fixture class name.</summary>
*)
{attribute 'monitoring' := 'call'}
PROPERTY ClassName : REFERENCE TO STRING
GET
ClassName REF= _ClassName;
END_GET
END_PROPERTY

(*!
<summary>Returns one fixed hash for all supported values, or raises the configured hash failure.</summary>
<description>
Equal values therefore always have equal hashes. This fixture intentionally sacrifices distribution.
</description>
*)
METHOD GetValueHashCode : UDINT
VAR_INPUT
	value : TOF_Core.GENERIC_VALUE;
END_VAR
IF ThrowOnHash THEN
	TOF_Core.Exceptions.ThrowStandard(
		sourceNamespaceName := NamespaceName,
		sourceClassName := ClassName,
		sourcePOUName := __POUNAME(),
		sourcePosition := __POSITION(),
		message := "Collection hash rejected"
	);
END_IF

GetValueHashCode := TOF_Core.UnsignedInt32.ZERO;
END_METHOD

(*!
<summary>Borrows the compiler-initialized test namespace.</summary>
*)
{attribute 'monitoring' := 'call'}
PROPERTY NamespaceName : REFERENCE TO STRING
GET
NamespaceName REF= CurrentNamespace.Name;
END_GET
END_PROPERTY

(*!
<summary>Reports the complete fixture instance size, excluding separately allocated storage.</summary>
*)
{attribute 'monitoring' := 'call'}
PROPERTY SelfSize : ULINT
GET
SelfSize := XSIZEOF(THIS^);
END_GET
END_PROPERTY

END_FUNCTION_BLOCK

// ---- Tests/Collections/Contract/CollectionPredicateProbe.TcPOU
(*
SPDX-FileCopyrightText: © 2026 Oleksandr Tiutyk <trofimich@gmail.com>
SPDX-License-Identifier: MIT
License: https://opensource.org/license/mit
*)

(*!
<summary>Matches every borrowed value until a configured callback count raises.</summary>
<description>
Counts callbacks without retaining operands. Used to prove skip/limit behavior and partial removal state.
</description>
*)

FUNCTION_BLOCK CollectionPredicateProbe EXTENDS TOF_Core.Object IMPLEMENTS TOF_Core.IPredicate
VAR_INPUT
	//! <summary>One-based callback number that raises; zero disables injection.</summary>
	ThrowOnCall : UDINT;
END_VAR
VAR_OUTPUT
	//! <summary>Number of Check callbacks since ResetCount.</summary>
	CallCount : UDINT;
END_VAR
VAR_STAT
	_ClassName : STRING := __POUNAME();
END_VAR

(*!
<summary>Counts the callback and returns TRUE unless this call is selected to raise.</summary>
*)
METHOD Check : BOOL
VAR_INPUT
	valueToCompare : __SYSTEM.AnyType;
END_VAR
CallCount := CallCount + 1;

IF ThrowOnCall <> TOF_Core.UnsignedInt32.ZERO AND_THEN CallCount = ThrowOnCall THEN
	TOF_Core.Exceptions.ThrowStandard(
		sourceNamespaceName := NamespaceName,
		sourceClassName := ClassName,
		sourcePOUName := __POUNAME(),
		sourcePosition := __POSITION(),
		message := "Collection predicate rejected"
	);
END_IF

Check := TRUE;
END_METHOD

(*!
<summary>Provides the concrete test fixture class name.</summary>
*)
{attribute 'monitoring' := 'call'}
PROPERTY ClassName : REFERENCE TO STRING
GET
ClassName REF= _ClassName;
END_GET
END_PROPERTY

(*!
<summary>Borrows the compiler-initialized test namespace.</summary>
*)
{attribute 'monitoring' := 'call'}
PROPERTY NamespaceName : REFERENCE TO STRING
GET
NamespaceName REF= CurrentNamespace.Name;
END_GET
END_PROPERTY

(*!
<summary>Resets only the observed callback count.</summary>
*)
METHOD ResetCount
CallCount := TOF_Core.UnsignedInt32.ZERO;
END_METHOD

(*!
<summary>Reports the complete fixture instance size, excluding separately allocated storage.</summary>
*)
{attribute 'monitoring' := 'call'}
PROPERTY SelfSize : ULINT
GET
SelfSize := XSIZEOF(THIS^);
END_GET
END_PROPERTY

END_FUNCTION_BLOCK

// ---- Tests/Collections/Contract/CollectionComparerProbe.TcPOU
(*
SPDX-FileCopyrightText: © 2026 Oleksandr Tiutyk <trofimich@gmail.com>
SPDX-License-Identifier: MIT
License: https://opensource.org/license/mit
*)

(*!
<summary>Counts generic ordering comparisons and raises at a configured call.</summary>
<description>
Operands remain borrowed and unchanged. Default generic ordering is used before and after injection.
</description>
*)

FUNCTION_BLOCK CollectionComparerProbe EXTENDS TOF_Core.Object IMPLEMENTS TOF_Core.IComparer
VAR_INPUT
	//! <summary>One-based comparison number that raises; zero disables injection.</summary>
	ThrowOnCall : UDINT;
END_VAR
VAR_OUTPUT
	//! <summary>Number of comparisons since ResetCount.</summary>
	CallCount : UDINT;
END_VAR
VAR_STAT
	_ClassName : STRING := __POUNAME();
END_VAR

(*!
<summary>Provides the concrete test fixture class name.</summary>
*)
{attribute 'monitoring' := 'call'}
PROPERTY ClassName : REFERENCE TO STRING
GET
ClassName REF= _ClassName;
END_GET
END_PROPERTY

(*!
<summary>Compares compatible borrowed values or raises on the selected callback.</summary>
*)
METHOD Compare : TOF_Core.COMPARISON_RESULT
VAR_INPUT
	first : TOF_Core.GENERIC_VALUE;
	second : TOF_Core.GENERIC_VALUE;
END_VAR
CallCount := CallCount + 1;

IF ThrowOnCall <> TOF_Core.UnsignedInt32.ZERO AND_THEN CallCount = ThrowOnCall THEN
	TOF_Core.Exceptions.ThrowStandard(
		sourceNamespaceName := NamespaceName,
		sourceClassName := ClassName,
		sourcePOUName := __POUNAME(),
		sourcePosition := __POSITION(),
		message := "Collection comparer rejected"
	);
END_IF

Compare := first.CompareTo(otherValue := second);
END_METHOD

(*!
<summary>Borrows the compiler-initialized test namespace.</summary>
*)
{attribute 'monitoring' := 'call'}
PROPERTY NamespaceName : REFERENCE TO STRING
GET
NamespaceName REF= CurrentNamespace.Name;
END_GET
END_PROPERTY

(*!
<summary>Resets only the observed comparison count.</summary>
*)
METHOD ResetCount
CallCount := TOF_Core.UnsignedInt32.ZERO;
END_METHOD

(*!
<summary>Reports the complete fixture instance size, excluding separately allocated storage.</summary>
*)
{attribute 'monitoring' := 'call'}
PROPERTY SelfSize : ULINT
GET
SelfSize := XSIZEOF(THIS^);
END_GET
END_PROPERTY

END_FUNCTION_BLOCK

// ---- Tests/Collections/Contract/CollectionsContractTestCase.TcPOU
(*
SPDX-FileCopyrightText: © 2026 Oleksandr Tiutyk <trofimich@gmail.com>
SPDX-License-Identifier: MIT
License: https://opensource.org/license/mit
*)

(*!
<summary>Runs one contract scenario and reports its own result.</summary>
<description>
Borrows the group fixture. The owning group serializes its cases in one task. AfterTest clears the fixture
after a successful run or an interrupted scenario. Terminal allocation failure uses the task boundary.
</description>
*)

{attribute 'no_assign'}
{attribute 'no_explicit_call' := 'do not call this function block directly'}
FUNCTION_BLOCK CollectionsContractTestCase EXTENDS TOF_Testing.SingleCycleTest
VAR_STAT
	{attribute 'hide'}
	_ClassName : STRING := __POUNAME();
END_VAR
VAR
	_Fixture : REFERENCE TO CollectionsContractTestFixture;
	_Scenario : COLLECTIONS_CONTRACT_SCENARIO;
END_VAR

(*!
<summary>Binds the group fixture and selects this case scenario.</summary>
<description>
Stores a borrowed reference without invoking the fixture. The owning group keeps it alive and
serializes use. TestElement initializes the name and parent.
</description>
<param name="name">Display name of this case.</param>
<param name="parent">Owning group.</param>
<param name="fixture">Live fixture owned by the group.</param>
<param name="scenario">Scenario assigned to this case.</param>
*)
METHOD FB_init : BOOL
VAR_INPUT
	bInitRetains: BOOL; // TRUE: the retain variables are initialized (reset warm / reset cold)
	bInCopyCode: BOOL; // TRUE: the instance will be copied to the copy code afterward (online change)
	name : WSTRING;
	parent : TOF_Testing.ITestElement;
	fixture : REFERENCE TO CollectionsContractTestFixture;
	scenario : COLLECTIONS_CONTRACT_SCENARIO;
END_VAR
IF NOT bInCopyCode THEN
	_Fixture REF= fixture;
	_Scenario := scenario;
END_IF

FB_init := TRUE;
END_METHOD

(*!
<summary>Runs the chosen scenario with the current assertions.</summary>
<description>
The fixture stays available to AfterTest if a call interrupts the scenario.
</description>
*)
METHOD PROTECTED ExecuteTest
VAR
	assertions : REFERENCE TO TOF_Testing.Assertions;
END_VAR
IF NOT __ISVALIDREF(_Fixture) THEN
	RecordFailure(message := "Missing collection contract fixture");

	RETURN;
END_IF

assertions REF= Assert;
_Fixture.ExecuteScenario(scenario := _Scenario, assertions := assertions);
END_METHOD

(*!
<summary>Clears the shared fixture and reports failed checked releases.</summary>
<description>
The fixture releases cursors before their sources. Cleanup preserves the first test failure and logs
any subsequent disposal failure.
</description>
*)
METHOD PROTECTED AfterTest
IF NOT __ISVALIDREF(_Fixture) THEN
	RETURN;
END_IF

IF NOT _Fixture.FinishScenario() THEN
	IF Outcome = TOF_Testing.TEST_OUTCOME.FAILED THEN
		Tc2_System.ADSLOGSTR(
			msgCtrlMask := Tc2_System.Global_Variables.ADSLOG_MSGTYPE_ERROR,
			msgFmtStr := 'Collection contract fixture cleanup failed in %s',
			strArg := TO_STRING(Name)
		);
	ELSE
		RecordFailure(message := "Collection contract fixture cleanup failed");
	END_IF
END_IF
END_METHOD

//! <summary>Borrows the concrete class name. Callers must not modify it.</summary>
{attribute 'monitoring' := 'call'}
PROPERTY ClassName : REFERENCE TO STRING
GET
ClassName REF= _ClassName;
END_GET
END_PROPERTY

//! <summary>Borrows the compiler-initialized namespace name. Callers must not modify it.</summary>
{attribute 'monitoring' := 'call'}
PROPERTY NamespaceName : REFERENCE TO STRING
GET
NamespaceName REF= CurrentNamespace.Name;
END_GET
END_PROPERTY

//! <summary>Reports the concrete instance size in bytes.</summary>
{attribute 'monitoring' := 'call'}
PROPERTY SelfSize : ULINT
GET
SelfSize := XSIZEOF(THIS^);
END_GET
END_PROPERTY

END_FUNCTION_BLOCK

// ---- Tests/Devices/IO/IOModelsTestGroup.TcPOU
(*
SPDX-FileCopyrightText: © 2026 Oleksandr Tiutyk <trofimich@gmail.com>
SPDX-License-Identifier: MIT
License: https://opensource.org/license/mit
*)

(*!
<summary>Groups PDO representation and simulated analog input binding scenarios.</summary>
<description>
Owns ten persistent cases and their fixed child array. Borrows the runner field containing the interface to
the controller-owned model fixture. The runner, fixture and children share one task and lifetime.
The group must not be copied because its children are bound to this instance.
</description>
*)

{attribute 'no_assign'}
{attribute 'no_explicit_call' := 'do not call this function block directly'}
FUNCTION_BLOCK IOModelsTestGroup EXTENDS TOF_Testing.TestGroup<10> IMPLEMENTS IIOModelsTestFixture
VAR_STAT
	{attribute 'hide'}
	_ClassName : STRING := __POUNAME();
END_VAR
VAR
	_FixtureSlot : POINTER TO IIOModelsTestFixture;
END_VAR
VAR
	_PulseTrain : IOModelsTestCase(
		name := "testPulseTrain",
		parent := THIS^,
		fixture := THIS^,
		scenario := IO_MODELS_TEST_SCENARIO.PULSE_TRAIN
	);
	_EncoderChannels : IOModelsTestCase(
		name := "testEncoderChannels",
		parent := THIS^,
		fixture := THIS^,
		scenario := IO_MODELS_TEST_SCENARIO.ENCODER_CHANNELS
	);
	_PowerMeasurement : IOModelsTestCase(
		name := "testPowerMeasurement",
		parent := THIS^,
		fixture := THIS^,
		scenario := IO_MODELS_TEST_SCENARIO.POWER_MEASUREMENT
	);
	_Auxiliary : IOModelsTestCase(
		name := "testAuxiliary",
		parent := THIS^,
		fixture := THIS^,
		scenario := IO_MODELS_TEST_SCENARIO.AUXILIARY
	);
	_CounterAndLoad : IOModelsTestCase(
		name := "testCounterAndLoad",
		parent := THIS^,
		fixture := THIS^,
		scenario := IO_MODELS_TEST_SCENARIO.COUNTER_AND_LOAD
	);
	_SerialAndDiagnostics : IOModelsTestCase(
		name := "testSerialAndDiagnostics",
		parent := THIS^,
		fixture := THIS^,
		scenario := IO_MODELS_TEST_SCENARIO.SERIAL_AND_DIAGNOSTICS
	);
	_DiscreteCatalog : IOModelsTestCase(
		name := "testDiscreteCatalog",
		parent := THIS^,
		fixture := THIS^,
		scenario := IO_MODELS_TEST_SCENARIO.DISCRETE_CATALOG
	);
	_AnalogRepresentations : IOModelsTestCase(
		name := "testAnalogRepresentations",
		parent := THIS^,
		fixture := THIS^,
		scenario := IO_MODELS_TEST_SCENARIO.ANALOG_REPRESENTATIONS
	);
	_DintBinding : IOModelsTestCase(
		name := "testDintBinding",
		parent := THIS^,
		fixture := THIS^,
		scenario := IO_MODELS_TEST_SCENARIO.DINT_BINDING
	);
	_RealBinding : IOModelsTestCase(
		name := "testRealBinding",
		parent := THIS^,
		fixture := THIS^,
		scenario := IO_MODELS_TEST_SCENARIO.REAL_BINDING
	);
END_VAR
VAR
	_Children : ARRAY [0.._ChildCount - 1] OF TOF_Testing.ITestElement :=
	[
		_PulseTrain,
		_EncoderChannels,
		_PowerMeasurement,
		_Auxiliary,
		_CounterAndLoad,
		_SerialAndDiagnostics,
		_DiscreteCatalog,
		_AnalogRepresentations,
		_DintBinding,
		_RealBinding
	];
END_VAR

(*!
<summary>Stores the address of the runner-owned fixture slot.</summary>
<description>Does not read the slot during initialization. The slot stays alive until after the group exits.</description>
<param name="name">Display name of the group.</param>
<param name="parent">Owning group or zero for a runner root.</param>
<param name="fixtureSlot">Address of the stable variable holding the controller fixture interface.</param>
*)
METHOD FB_init : BOOL
VAR_INPUT
	bInitRetains: BOOL; // TRUE: the retain variables are initialized (reset warm / reset cold)
	bInCopyCode: BOOL; // TRUE: the instance will be copied to the copy code afterward (online change)
	name : WSTRING;
	parent : TOF_Testing.ITestElement;
	fixtureSlot : POINTER TO IIOModelsTestFixture;
END_VAR
IF NOT bInCopyCode THEN
	_FixtureSlot := fixtureSlot;
END_IF

FB_init := TRUE;
END_METHOD

(*!
<summary>Runs one IO model scenario and reports to the current case.</summary>
<description>Use from the owning test task. The fixture never retains assertions.</description>
<param name="scenario">Scenario assigned to the caller.</param>
<param name="assertions">Valid assertion context borrowed from the active case.</param>
*)
METHOD ExecuteScenario
VAR_INPUT
	scenario : IO_MODELS_TEST_SCENARIO;
	assertions : REFERENCE TO TOF_Testing.Assertions;
END_VAR
VAR
	fixture : IIOModelsTestFixture;
END_VAR
IF _FixtureSlot <> 0 THEN
	fixture := _FixtureSlot^;
END_IF

IF fixture = 0 THEN
	assertions.ThatBool(actual := FALSE, message := "Missing IO model fixture").IsTrue();

	RETURN;
END_IF

fixture.ExecuteScenario(scenario := scenario, assertions := assertions);
END_METHOD

(*!
<summary>Borrows the persistent case array. Callers must not modify it.</summary>
*)
{attribute 'monitoring' := 'call'}
PROPERTY Children : REFERENCE TO ARRAY [0.._ChildCount - 1] OF TOF_Testing.ITestElement
GET
Children REF= _Children;
END_GET
END_PROPERTY

(*!
<summary>Borrows the concrete class name. Callers must not modify it.</summary>
*)
{attribute 'monitoring' := 'call'}
PROPERTY ClassName : REFERENCE TO STRING
GET
ClassName REF= _ClassName;
END_GET
END_PROPERTY

(*!
<summary>Borrows the project namespace name. Callers must not modify it.</summary>
*)
{attribute 'monitoring' := 'call'}
PROPERTY NamespaceName : REFERENCE TO STRING
GET
NamespaceName REF= CurrentNamespace.Name;
END_GET
END_PROPERTY

(*!
<summary>Reports the complete instance size in bytes.</summary>
*)
{attribute 'monitoring' := 'call'}
PROPERTY SelfSize : ULINT
GET
SelfSize := XSIZEOF(THIS^);
END_GET
END_PROPERTY

END_FUNCTION_BLOCK

// ---- Tests/Devices/IO/IOModelsTestCase.TcPOU
(*
SPDX-FileCopyrightText: © 2026 Oleksandr Tiutyk <trofimich@gmail.com>
SPDX-License-Identifier: MIT
License: https://opensource.org/license/mit
*)

(*!
<summary>Runs one IO model scenario and reports its own outcome.</summary>
<description>Borrows its group as the scenario provider. Use the group and its cases from a single task.</description>
*)

{attribute 'no_assign'}
{attribute 'no_explicit_call' := 'do not call this function block directly'}
FUNCTION_BLOCK IOModelsTestCase EXTENDS TOF_Testing.SingleCycleTest
VAR_STAT
	{attribute 'hide'}
	_ClassName : STRING := __POUNAME();
END_VAR
VAR
	_Fixture : IIOModelsTestFixture;
	_Scenario : IO_MODELS_TEST_SCENARIO;
END_VAR

(*!
<summary>Stores the case scenario and its borrowed provider without invoking it.</summary>
<param name="name">Name reported for the individual case.</param>
<param name="parent">Group that owns this case.</param>
<param name="fixture">Scenario provider that outlives the case.</param>
<param name="scenario">Scenario selected for the case.</param>
*)
METHOD FB_init : BOOL
VAR_INPUT
	bInitRetains: BOOL; // TRUE: the retain variables are initialized (reset warm / reset cold)
	bInCopyCode: BOOL; // TRUE: the instance will be copied to the copy code afterward (online change)
	name : WSTRING;
	parent : TOF_Testing.ITestElement;
	fixture : IIOModelsTestFixture;
	scenario : IO_MODELS_TEST_SCENARIO;
END_VAR
IF NOT bInCopyCode THEN
	_Fixture := fixture;
	_Scenario := scenario;
END_IF

FB_init := TRUE;
END_METHOD

(*!
<summary>Executes the selected scenario using the assertion context of this run.</summary>
*)
METHOD PROTECTED ExecuteTest
VAR
	assertions : REFERENCE TO TOF_Testing.Assertions;
END_VAR
IF _Fixture = 0 THEN
	RecordFailure(message := "Missing IO model scenario provider");

	RETURN;
END_IF

assertions REF= Assert;
_Fixture.ExecuteScenario(scenario := _Scenario, assertions := assertions);
END_METHOD

(*!
<summary>Borrows the concrete class name. Callers must not modify it.</summary>
*)
{attribute 'monitoring' := 'call'}
PROPERTY ClassName : REFERENCE TO STRING
GET
ClassName REF= _ClassName;
END_GET
END_PROPERTY

(*!
<summary>Borrows the project namespace name. Callers must not modify it.</summary>
*)
{attribute 'monitoring' := 'call'}
PROPERTY NamespaceName : REFERENCE TO STRING
GET
NamespaceName REF= CurrentNamespace.Name;
END_GET
END_PROPERTY

(*!
<summary>Reports the complete instance size in bytes.</summary>
*)
{attribute 'monitoring' := 'call'}
PROPERTY SelfSize : ULINT
GET
SelfSize := XSIZEOF(THIS^);
END_GET
END_PROPERTY

END_FUNCTION_BLOCK

// ---- Tests/Workflow/WorkflowComprehensiveTestGroup.TcPOU
(*
SPDX-FileCopyrightText: © 2026 Oleksandr Tiutyk <trofimich@gmail.com>
SPDX-License-Identifier: MIT
License: https://opensource.org/license/mit
*)

(*!
<summary>Groups workflow scenario, comparisons, lifecycle and variable-scope tests.</summary>
<description>Owns the fixed case tree and runs its leaves in order in the controller task.</description>
*)

{attribute 'no_assign'}
{attribute 'no_explicit_call' := 'do not call this function block directly'}
FUNCTION_BLOCK WorkflowComprehensiveTestGroup EXTENDS TOF_Testing.TestGroup<14>
VAR_STAT
	{attribute 'hide'}
	_ClassName : STRING := __POUNAME();
END_VAR
VAR
	_EndToEndComprehensiveScenario : WorkflowComprehensiveTestCase(
		name := "TestEndToEndComprehensiveScenario",
		parent := THIS^,
		scenario := WORKFLOW_COMPREHENSIVE_TEST_SCENARIO.END_TO_END_COMPREHENSIVE_SCENARIO
	);
	_WorkflowReset : WorkflowComprehensiveTestCase(
		name := "TestWorkflowReset",
		parent := THIS^,
		scenario := WORKFLOW_COMPREHENSIVE_TEST_SCENARIO.WORKFLOW_RESET
	);
	_WorkflowCancel : WorkflowComprehensiveTestCase(
		name := "TestWorkflowCancel",
		parent := THIS^,
		scenario := WORKFLOW_COMPREHENSIVE_TEST_SCENARIO.WORKFLOW_CANCEL
	);
	_ParallelActivityWaitAll : WorkflowComprehensiveTestCase(
		name := "TestParallelActivityWaitAll",
		parent := THIS^,
		scenario := WORKFLOW_COMPREHENSIVE_TEST_SCENARIO.PARALLEL_ACTIVITY_WAIT_ALL
	);
	_ParallelActivityWaitAny : WorkflowComprehensiveTestCase(
		name := "TestParallelActivityWaitAny",
		parent := THIS^,
		scenario := WORKFLOW_COMPREHENSIVE_TEST_SCENARIO.PARALLEL_ACTIVITY_WAIT_ANY
	);
	_NotCondition : WorkflowComprehensiveTestCase(
		name := "TestNotCondition",
		parent := THIS^,
		scenario := WORKFLOW_COMPREHENSIVE_TEST_SCENARIO.NOT_CONDITION
	);
	_CompareVariableCondition : WorkflowComprehensiveTestCase(
		name := "TestCompareVariableCondition",
		parent := THIS^,
		scenario := WORKFLOW_COMPREHENSIVE_TEST_SCENARIO.COMPARE_VARIABLE_CONDITION
	);
	_MixedNumericComparison : WorkflowComprehensiveTestCase(
		name := "TestMixedNumericComparison",
		parent := THIS^,
		scenario := WORKFLOW_COMPREHENSIVE_TEST_SCENARIO.MIXED_NUMERIC_COMPARISON
	);
	_MixedTextComparison : WorkflowComprehensiveTestCase(
		name := "TestMixedTextComparison",
		parent := THIS^,
		scenario := WORKFLOW_COMPREHENSIVE_TEST_SCENARIO.MIXED_TEXT_COMPARISON
	);
	_StandardComparisonFallback : WorkflowComprehensiveTestCase(
		name := "TestStandardComparisonFallback",
		parent := THIS^,
		scenario := WORKFLOW_COMPREHENSIVE_TEST_SCENARIO.STANDARD_COMPARISON_FALLBACK
	);
	_IncompatibleComparisonPairs : WorkflowComprehensiveTestCase(
		name := "TestIncompatibleComparisonPairs",
		parent := THIS^,
		scenario := WORKFLOW_COMPREHENSIVE_TEST_SCENARIO.INCOMPATIBLE_COMPARISON_PAIRS
	);
	_DirectWorkflowDynamicCreation : WorkflowComprehensiveTestCase(
		name := "TestDirectWorkflowDynamicCreation",
		parent := THIS^,
		scenario := WORKFLOW_COMPREHENSIVE_TEST_SCENARIO.DIRECT_WORKFLOW_DYNAMIC_CREATION
	);
	_ActivityVariableScopingAndShadowing : WorkflowComprehensiveTestCase(
		name := "TestActivityVariableScopingAndShadowing",
		parent := THIS^,
		scenario := WORKFLOW_COMPREHENSIVE_TEST_SCENARIO.ACTIVITY_VARIABLE_SCOPING_AND_SHADOWING
	);
	_VariableRegistrationValidation : WorkflowComprehensiveTestCase(
		name := "TestVariableRegistrationValidation",
		parent := THIS^,
		scenario := WORKFLOW_COMPREHENSIVE_TEST_SCENARIO.VARIABLE_REGISTRATION_VALIDATION
	);
END_VAR
VAR
	_Children : ARRAY [0.._ChildCount - 1] OF TOF_Testing.ITestElement :=
	[
		_EndToEndComprehensiveScenario,
		_WorkflowReset,
		_WorkflowCancel,
		_ParallelActivityWaitAll,
		_ParallelActivityWaitAny,
		_NotCondition,
		_CompareVariableCondition,
		_MixedNumericComparison,
		_MixedTextComparison,
		_StandardComparisonFallback,
		_IncompatibleComparisonPairs,
		_DirectWorkflowDynamicCreation,
		_ActivityVariableScopingAndShadowing,
		_VariableRegistrationValidation
	];
END_VAR

(*!
<summary>Borrows the persistent case array. Callers must not modify it.</summary>
*)
{attribute 'monitoring' := 'call'}
PROPERTY Children : REFERENCE TO ARRAY [0.._ChildCount - 1] OF TOF_Testing.ITestElement
GET
Children REF= _Children;
END_GET
END_PROPERTY

(*!
<summary>Borrows the concrete class name. Callers must not modify it.</summary>
*)
{attribute 'monitoring' := 'call'}
PROPERTY ClassName : REFERENCE TO STRING
GET
ClassName REF= _ClassName;
END_GET
END_PROPERTY

(*!
<summary>Borrows the project namespace name. Callers must not modify it.</summary>
*)
{attribute 'monitoring' := 'call'}
PROPERTY NamespaceName : REFERENCE TO STRING
GET
NamespaceName REF= CurrentNamespace.Name;
END_GET
END_PROPERTY

(*!
<summary>Reports the complete instance size in bytes.</summary>
*)
{attribute 'monitoring' := 'call'}
PROPERTY SelfSize : ULINT
GET
SelfSize := XSIZEOF(THIS^);
END_GET
END_PROPERTY

END_FUNCTION_BLOCK

// ---- Tests/Workflow/WorkflowComprehensiveTestCase.TcPOU
(*
SPDX-FileCopyrightText: © 2026 Oleksandr Tiutyk <trofimich@gmail.com>
SPDX-License-Identifier: MIT
License: https://opensource.org/license/mit
*)

(*!
<summary>Runs one workflow integration scenario in an isolated fixture.</summary>
<description>
Owns a freshly allocated fixture for the active run. AfterTest releases it after success or a reported
exception. A concrete pointer preserves FB_exit for the fixture and its nested resource owners.
Use one task. Do not copy the test case while it owns a fixture.
</description>
*)

{attribute 'no_assign'}
{attribute 'no_explicit_call' := 'do not call this function block directly'}
FUNCTION_BLOCK WorkflowComprehensiveTestCase EXTENDS TOF_Testing.SingleCycleTest
VAR_STAT
	{attribute 'hide'}
	_ClassName : STRING := __POUNAME();
END_VAR
VAR
	_Scenario : WORKFLOW_COMPREHENSIVE_TEST_SCENARIO;
	_Fixture : POINTER TO WorkflowComprehensiveTestFixture;
END_VAR

(*!
<summary>Selects the scenario without allocating its fixture.</summary>
<param name="name">Name reported for this case.</param>
<param name="parent">Group that owns this case.</param>
<param name="scenario">Scenario selected for the case.</param>
*)
METHOD FB_init : BOOL
VAR_INPUT
	bInitRetains: BOOL; // TRUE: the retain variables are initialized (reset warm / reset cold)
	bInCopyCode: BOOL; // TRUE: the instance will be copied to the copy code afterward (online change)
	name : WSTRING;
	parent : TOF_Testing.ITestElement;
	scenario : WORKFLOW_COMPREHENSIVE_TEST_SCENARIO;
END_VAR
IF NOT bInCopyCode THEN
	_Scenario := scenario;
END_IF

FB_init := TRUE;
END_METHOD

(*!
<summary>Allocates a fresh fixture and runs the selected scenario.</summary>
<description>Terminal allocation failure is raised at the task boundary after case handling.</description>
*)
METHOD PROTECTED ExecuteTest
VAR
	assertions : REFERENCE TO TOF_Testing.Assertions;
END_VAR
_Fixture := __NEW(WorkflowComprehensiveTestFixture);

IF _Fixture = 0 THEN
	TOF_Core.DynamicMemoryManager.RaiseAllocationFailure();

	RETURN;
END_IF

assertions REF= Assert;
_Fixture^.ExecuteScenario(scenario := _Scenario, assertions := assertions);
END_METHOD

(*!
<summary>Releases the fixture before the case outcome is published.</summary>
<description>The framework records an exception from teardown. Clear the stored alias before releasing.</description>
*)
METHOD PROTECTED AfterTest
VAR
	fixture : POINTER TO WorkflowComprehensiveTestFixture;
END_VAR
fixture := _Fixture;
_Fixture := 0;

IF fixture <> 0 THEN
	__DELETE(fixture);
END_IF
END_METHOD

(*!
<summary>Releases an active fixture if the case is unloaded before its teardown.</summary>
<description>The fixture and its nested FB_exit paths complete without exceptions.</description>
<param name="bInCopyCode">TwinCAT copy-code exit marker. The previous instance leaves copied storage alive.</param>
*)
METHOD FB_exit : BOOL
VAR_INPUT
	bInCopyCode : BOOL;
END_VAR
IF NOT bInCopyCode AND_THEN _Fixture <> 0 THEN
	__DELETE(_Fixture);
END_IF

FB_exit := TRUE;
END_METHOD

(*!
<summary>Borrows the concrete class name. Callers must not modify it.</summary>
*)
{attribute 'monitoring' := 'call'}
PROPERTY ClassName : REFERENCE TO STRING
GET
ClassName REF= _ClassName;
END_GET
END_PROPERTY

(*!
<summary>Borrows the project namespace name. Callers must not modify it.</summary>
*)
{attribute 'monitoring' := 'call'}
PROPERTY NamespaceName : REFERENCE TO STRING
GET
NamespaceName REF= CurrentNamespace.Name;
END_GET
END_PROPERTY

(*!
<summary>Reports the complete instance size in bytes.</summary>
*)
{attribute 'monitoring' := 'call'}
PROPERTY SelfSize : ULINT
GET
SelfSize := XSIZEOF(THIS^);
END_GET
END_PROPERTY

END_FUNCTION_BLOCK

// ---- Tests/Workflow/WorkflowComprehensiveTestFixture.TcPOU
(*
SPDX-FileCopyrightText: © 2026 Oleksandr Tiutyk <trofimich@gmail.com>
SPDX-License-Identifier: MIT
License: https://opensource.org/license/mit
*)

(*!
<summary>Owns the state used by one workflow integration test scenario.</summary>
<description>
Each fixture starts with freshly constructed function blocks and stores no borrowed assertion context.
Workflows own their dynamically registered nodes. The direct-creation case also tracks its concrete pointer
until explicit deletion or fixture teardown. Tasks and delay inputs are self-contained PLC simulations.
</description>
*)

{attribute 'enable_dynamic_creation'}
{attribute 'no_assign'}
{attribute 'no_explicit_call' := 'do not call this function block directly'}
FUNCTION_BLOCK WorkflowComprehensiveTestFixture
VAR_STAT
	//! <summary>Class name shared by all instances of this function block.</summary>
	{attribute 'hide'}
	_ClassName : STRING := __POUNAME();
END_VAR
VAR
	_Workflow : ComprehensiveTestWorkflow;
	//! <summary>Owns the comparison condition and its reference snapshot throughout the suite lifetime.</summary>
	_ComparisonCondition : TOF_Workflow.CompareVariableCondition(workflow := _Workflow);

	//! <summary>Owns isolated pair-comparison configuration and borrowed bindings to the following fixtures.</summary>
	_PairComparisonCondition : TOF_Workflow.CompareVariableCondition(workflow := 0);
	_ComparisonNarrowInteger : SINT := 127;
	_ComparisonWideInteger : LINT := 128;
	_ComparisonSignedInteger : INT := -1;
	_ComparisonUnsignedInteger : UINT := TOF_Core.UnsignedInt16.MAX_VALUE;
	_ComparisonFloatingValue : LREAL;

	_ComparisonText : STRING(300);
	_ComparisonWideText : WSTRING(300);

	_FirstComparisonTimeOfDay : TIME_OF_DAY := TOD#08:00:00;
	_SecondComparisonTimeOfDay : TIME_OF_DAY := TOD#09:00:00;
	_FirstComparisonBytes : TOF_Core.REAL_UNION;
	_SecondComparisonBytes : TOF_Core.REAL_UNION;
	_ComparisonUnrelatedInteger : DINT;
	_ComparisonObject : TOF_Comparison.StorageAddressComparer;

	_ThrowingActivity : ThrowingTestActivity(workflow := _Workflow);
	_CounterTask : CounterTask(name := "CounterTask");

	_DynamicTestVar : DINT := 100;
	_WorkflowScopeVar : DINT := 200;
	_ParentScopeVar : DINT := 300;
	_ChildLocalVar : DINT := 400;

	//! <summary>Owns direct dynamic-creation coverage even when a test raises unexpectedly.</summary>
	_DirectWorkflow : POINTER TO TOF_Workflow.Workflow;

	_ResetWorkflow : ComprehensiveTestWorkflow;
	_ResetActivity : TOF_Workflow.DelayActivity(workflow := _ResetWorkflow);

	_ValidationWorkflow : TOF_Workflow.Workflow;
	_ValidationActivity : TOF_Workflow.DelayActivity(workflow := _ValidationWorkflow);
	_ValidationValue : DINT;

	_NotWorkflow : ComprehensiveTestWorkflow;
	_NotRoot : TOF_Workflow.DelayActivity(workflow := _NotWorkflow);
	_WaitAllWorkflow : TOF_Workflow.Workflow;
	_WaitAnyWorkflow : ComprehensiveTestWorkflow;
	_WaitAnyRoot : TOF_Workflow.DelayActivity(workflow := _WaitAnyWorkflow);
	_ScopeWorkflow : TOF_Workflow.Workflow;
END_VAR

(*!
<summary>Dispatches one scenario against the fresh fixture.</summary>
<description>Call once per fixture. Each method uses the assertions of the receiving case.</description>
<param name="scenario">Scenario assigned to the caller.</param>
<param name="assertions">Valid assertion context borrowed from the active case.</param>
*)
METHOD ExecuteScenario
VAR_INPUT
	scenario : WORKFLOW_COMPREHENSIVE_TEST_SCENARIO;
	assertions : REFERENCE TO TOF_Testing.Assertions;
END_VAR
CASE scenario OF
	WORKFLOW_COMPREHENSIVE_TEST_SCENARIO.END_TO_END_COMPREHENSIVE_SCENARIO:
		testEndToEndComprehensiveScenario(assertions := assertions);

	WORKFLOW_COMPREHENSIVE_TEST_SCENARIO.WORKFLOW_RESET:
		testWorkflowReset(assertions := assertions);

	WORKFLOW_COMPREHENSIVE_TEST_SCENARIO.WORKFLOW_CANCEL:
		testWorkflowCancel(assertions := assertions);

	WORKFLOW_COMPREHENSIVE_TEST_SCENARIO.PARALLEL_ACTIVITY_WAIT_ALL:
		testParallelActivityWaitAll(assertions := assertions);

	WORKFLOW_COMPREHENSIVE_TEST_SCENARIO.PARALLEL_ACTIVITY_WAIT_ANY:
		testParallelActivityWaitAny(assertions := assertions);

	WORKFLOW_COMPREHENSIVE_TEST_SCENARIO.NOT_CONDITION:
		testNotCondition(assertions := assertions);

	WORKFLOW_COMPREHENSIVE_TEST_SCENARIO.COMPARE_VARIABLE_CONDITION:
		testCompareVariableCondition(assertions := assertions);

	WORKFLOW_COMPREHENSIVE_TEST_SCENARIO.MIXED_NUMERIC_COMPARISON:
		testMixedNumericComparison(assertions := assertions);

	WORKFLOW_COMPREHENSIVE_TEST_SCENARIO.MIXED_TEXT_COMPARISON:
		testMixedTextComparison(assertions := assertions);

	WORKFLOW_COMPREHENSIVE_TEST_SCENARIO.STANDARD_COMPARISON_FALLBACK:
		testStandardComparisonFallback(assertions := assertions);

	WORKFLOW_COMPREHENSIVE_TEST_SCENARIO.INCOMPATIBLE_COMPARISON_PAIRS:
		testIncompatibleComparisonPairs(assertions := assertions);

	WORKFLOW_COMPREHENSIVE_TEST_SCENARIO.DIRECT_WORKFLOW_DYNAMIC_CREATION:
		testDirectWorkflowDynamicCreation(assertions := assertions);

	WORKFLOW_COMPREHENSIVE_TEST_SCENARIO.ACTIVITY_VARIABLE_SCOPING_AND_SHADOWING:
		testActivityVariableScopingAndShadowing(assertions := assertions);

	WORKFLOW_COMPREHENSIVE_TEST_SCENARIO.VARIABLE_REGISTRATION_VALIDATION:
		testVariableRegistrationValidation(assertions := assertions);
ELSE
	assertions.ThatBool(actual := FALSE, message := "Unknown workflow integration scenario").IsTrue();
END_CASE
END_METHOD

(*!
<summary>Borrows the concrete class name. Callers must not modify it.</summary>
*)
{attribute 'monitoring' := 'call'}
PROPERTY ClassName : REFERENCE TO STRING
GET
ClassName REF= _ClassName;
END_GET
END_PROPERTY

(*!
<summary>Borrows the project namespace name. Callers must not modify it.</summary>
*)
{attribute 'monitoring' := 'call'}
PROPERTY NamespaceName : REFERENCE TO STRING
GET
NamespaceName REF= CurrentNamespace.Name;
END_GET
END_PROPERTY

(*!
<summary>Builds the registered scenario tree with allocation guards before every dereference.</summary>
<description>Registered nodes remain workflow-owned if a later configuration operation raises.</description>
*)
METHOD PRIVATE buildScenarioTree
VAR
	rootSequence : POINTER TO TOF_Workflow.SequenceActivity;
	initBatchTarget : POINTER TO TOF_Workflow.AssignVariableActivity;

	parallelStep : POINTER TO TOF_Workflow.ParallelActivity;
	parallelDelay : POINTER TO TOF_Workflow.DelayActivity;
	parallelAssign : POINTER TO TOF_Workflow.AssignVariableActivity;

	whileCondition : POINTER TO TOF_Workflow.VariableHasValueCondition;
	whileActivity : POINTER TO TOF_Workflow.WhileActivity;
	whileBody : POINTER TO TOF_Workflow.SequenceActivity;

	feedTaskActivity : POINTER TO TOF_Workflow.InvokeTaskActivity;

	condPart : POINTER TO TOF_Workflow.VariableHasValueCondition;
	condVacuum : POINTER TO TOF_Workflow.VariableHasValueCondition;
	compCond : POINTER TO TOF_Workflow.CompositeCondition;
	waitCondAct : POINTER TO TOF_Workflow.WaitConditionActivity;

	delayAct : POINTER TO TOF_Workflow.DelayActivity;

	pickAct : POINTER TO TOF_Workflow.WaitAndPickActivity;
	condOk : POINTER TO TOF_Workflow.VariableHasValueCondition;
	actOk : POINTER TO TOF_Workflow.AssignVariableActivity;
	condRej : POINTER TO TOF_Workflow.VariableHasValueCondition;
	actRej : POINTER TO TOF_Workflow.AssignVariableActivity;

	ifCond : POINTER TO TOF_Workflow.VariableHasValueCondition;
	trueAct : POINTER TO TOF_Workflow.DelayActivity;
	ifElseAct : POINTER TO TOF_Workflow.IfElseActivity;

	tryCatchAct : POINTER TO TOF_Workflow.TryCatchActivity;
	catchAct : POINTER TO RecoveryCatchTestActivity;

	refuseReason : TOF_Core.ERROR_MESSAGE;
	initTargetValue : INT := 2;
	producedIncrement : INT := 1;
	rejectIncrement : INT := 1;
	trueValue : BOOL := TRUE;
	falseValue : BOOL := FALSE;
	zeroCount : INT := 0;
END_VAR
// 1. Root Sequence
rootSequence := __NEW(TOF_Workflow.SequenceActivity(workflow := _Workflow));

IF rootSequence = 0 THEN
	TOF_Core.DynamicMemoryManager.RaiseAllocationFailure();
END_IF

_Workflow.RegisterChild(child := rootSequence^);

// 2. AssignVariableActivity: initialize BatchTarget
initBatchTarget := __NEW(TOF_Workflow.AssignVariableActivity(workflow := _Workflow));

IF initBatchTarget = 0 THEN
	TOF_Core.DynamicMemoryManager.RaiseAllocationFailure();
END_IF

_Workflow.RegisterChild(child := initBatchTarget^);
initBatchTarget^.Configure(targetVariableName := 'BatchTarget', value := initTargetValue);
rootSequence^.AddChildActivity(activity := initBatchTarget^);

// 2.5. ParallelActivity: concurrently run a delay and an assignment with WAIT_ALL
parallelStep := __NEW(TOF_Workflow.ParallelActivity(workflow := _Workflow));

IF parallelStep = 0 THEN
	TOF_Core.DynamicMemoryManager.RaiseAllocationFailure();
END_IF

_Workflow.RegisterChild(child := parallelStep^);
parallelStep^.Mode := TOF_Workflow.PARALLEL_JOIN_MODE.WAIT_ALL;

parallelDelay := __NEW(TOF_Workflow.DelayActivity(workflow := _Workflow));

IF parallelDelay = 0 THEN
	TOF_Core.DynamicMemoryManager.RaiseAllocationFailure();
END_IF

_Workflow.RegisterChild(child := parallelDelay^);
parallelDelay^.Interval := T#0S;
parallelStep^.AddChildActivity(activity := parallelDelay^);

parallelAssign := __NEW(TOF_Workflow.AssignVariableActivity(workflow := _Workflow));

IF parallelAssign = 0 THEN
	TOF_Core.DynamicMemoryManager.RaiseAllocationFailure();
END_IF

_Workflow.RegisterChild(child := parallelAssign^);
parallelAssign^.Configure(targetVariableName := 'SensorFeedPart', value := trueValue);
parallelStep^.AddChildActivity(activity := parallelAssign^);

rootSequence^.AddChildActivity(activity := parallelStep^);

// 3. WhileActivity: run while ProducedCount = 0
whileCondition := __NEW(TOF_Workflow.VariableHasValueCondition(workflow := _Workflow));

IF whileCondition = 0 THEN
	TOF_Core.DynamicMemoryManager.RaiseAllocationFailure();
END_IF

_Workflow.RegisterChild(child := whileCondition^);
whileCondition^.Configure(monitoredVariableName := 'ProducedCount', referenceValue := zeroCount);

whileActivity := __NEW(TOF_Workflow.WhileActivity(workflow := _Workflow));

IF whileActivity = 0 THEN
	TOF_Core.DynamicMemoryManager.RaiseAllocationFailure();
END_IF

_Workflow.RegisterChild(child := whileActivity^);

whileBody := __NEW(TOF_Workflow.SequenceActivity(workflow := _Workflow));

IF whileBody = 0 THEN
	TOF_Core.DynamicMemoryManager.RaiseAllocationFailure();
END_IF

_Workflow.RegisterChild(child := whileBody^);

whileActivity^.Configure(condition := whileCondition^, body := whileBody^);
rootSequence^.AddChildActivity(activity := whileActivity^);

// 3.1. InvokeTaskActivity inside while body
feedTaskActivity := __NEW(TOF_Workflow.InvokeTaskActivity(workflow := _Workflow));

IF feedTaskActivity = 0 THEN
	TOF_Core.DynamicMemoryManager.RaiseAllocationFailure();
END_IF

_Workflow.RegisterChild(child := feedTaskActivity^);
_CounterTask.Reset(refuseReason => refuseReason);
_CounterTask.TargetValue := 1;
feedTaskActivity^.Configure(task := _CounterTask);
whileBody^.AddChildActivity(activity := feedTaskActivity^);

// 3.2. WaitConditionActivity with CompositeCondition (AND)
condPart := __NEW(TOF_Workflow.VariableHasValueCondition(workflow := _Workflow));

IF condPart = 0 THEN
	TOF_Core.DynamicMemoryManager.RaiseAllocationFailure();
END_IF

_Workflow.RegisterChild(child := condPart^);
condPart^.Configure(monitoredVariableName := 'SensorFeedPart', referenceValue := trueValue);

condVacuum := __NEW(TOF_Workflow.VariableHasValueCondition(workflow := _Workflow));

IF condVacuum = 0 THEN
	TOF_Core.DynamicMemoryManager.RaiseAllocationFailure();
END_IF

_Workflow.RegisterChild(child := condVacuum^);
condVacuum^.Configure(monitoredVariableName := 'SensorVacuumOk', referenceValue := trueValue);

compCond := __NEW(TOF_Workflow.CompositeCondition(workflow := _Workflow));

IF compCond = 0 THEN
	TOF_Core.DynamicMemoryManager.RaiseAllocationFailure();
END_IF

_Workflow.RegisterChild(child := compCond^);
compCond^.LogicalOperator := TOF_Workflow.LOGICAL_OPERATOR.AND_;
compCond^.AddChildCondition(condition := condPart^);
compCond^.AddChildCondition(condition := condVacuum^);

waitCondAct := __NEW(TOF_Workflow.WaitConditionActivity(workflow := _Workflow));

IF waitCondAct = 0 THEN
	TOF_Core.DynamicMemoryManager.RaiseAllocationFailure();
END_IF

_Workflow.RegisterChild(child := waitCondAct^);
waitCondAct^.Configure(condition := compCond^);
whileBody^.AddChildActivity(activity := waitCondAct^);

// 3.3. DelayActivity
delayAct := __NEW(TOF_Workflow.DelayActivity(workflow := _Workflow));

IF delayAct = 0 THEN
	TOF_Core.DynamicMemoryManager.RaiseAllocationFailure();
END_IF

_Workflow.RegisterChild(child := delayAct^);
delayAct^.Interval := T#0S;
whileBody^.AddChildActivity(activity := delayAct^);

// 3.4. WaitAndPickActivity (Inspection decision)
pickAct := __NEW(TOF_Workflow.WaitAndPickActivity(workflow := _Workflow));

IF pickAct = 0 THEN
	TOF_Core.DynamicMemoryManager.RaiseAllocationFailure();
END_IF

_Workflow.RegisterChild(child := pickAct^);

condOk := __NEW(TOF_Workflow.VariableHasValueCondition(workflow := _Workflow));

IF condOk = 0 THEN
	TOF_Core.DynamicMemoryManager.RaiseAllocationFailure();
END_IF

_Workflow.RegisterChild(child := condOk^);
condOk^.Configure(monitoredVariableName := 'SensorInspectionOk', referenceValue := trueValue);

actOk := __NEW(TOF_Workflow.AssignVariableActivity(workflow := _Workflow));

IF actOk = 0 THEN
	TOF_Core.DynamicMemoryManager.RaiseAllocationFailure();
END_IF

_Workflow.RegisterChild(child := actOk^);
actOk^.Configure(targetVariableName := 'ProducedCount', value := producedIncrement);
pickAct^.AddBranch(condition := condOk^, activity := actOk^);

condRej := __NEW(TOF_Workflow.VariableHasValueCondition(workflow := _Workflow));

IF condRej = 0 THEN
	TOF_Core.DynamicMemoryManager.RaiseAllocationFailure();
END_IF

_Workflow.RegisterChild(child := condRej^);
condRej^.Configure(monitoredVariableName := 'SensorInspectionOk', referenceValue := falseValue);

actRej := __NEW(TOF_Workflow.AssignVariableActivity(workflow := _Workflow));

IF actRej = 0 THEN
	TOF_Core.DynamicMemoryManager.RaiseAllocationFailure();
END_IF

_Workflow.RegisterChild(child := actRej^);
actRej^.Configure(targetVariableName := 'RejectCount', value := rejectIncrement);
pickAct^.AddBranch(condition := condRej^, activity := actRej^);

whileBody^.AddChildActivity(activity := pickAct^);

// 3.5. IfElseActivity
ifCond := __NEW(TOF_Workflow.VariableHasValueCondition(workflow := _Workflow));

IF ifCond = 0 THEN
	TOF_Core.DynamicMemoryManager.RaiseAllocationFailure();
END_IF

_Workflow.RegisterChild(child := ifCond^);
ifCond^.Configure(monitoredVariableName := 'SensorInspectionOk', referenceValue := trueValue);

trueAct := __NEW(TOF_Workflow.DelayActivity(workflow := _Workflow));

IF trueAct = 0 THEN
	TOF_Core.DynamicMemoryManager.RaiseAllocationFailure();
END_IF

_Workflow.RegisterChild(child := trueAct^);
trueAct^.Interval := T#0S;

ifElseAct := __NEW(TOF_Workflow.IfElseActivity(workflow := _Workflow));

IF ifElseAct = 0 THEN
	TOF_Core.DynamicMemoryManager.RaiseAllocationFailure();
END_IF

_Workflow.RegisterChild(child := ifElseAct^);
ifElseAct^.Configure(condition := ifCond^, trueActivity := trueAct^, falseActivity := 0);
whileBody^.AddChildActivity(activity := ifElseAct^);

// 3.6. TryCatchActivity: verifies exception interception and recovery
tryCatchAct := __NEW(TOF_Workflow.TryCatchActivity(workflow := _Workflow));

IF tryCatchAct = 0 THEN
	TOF_Core.DynamicMemoryManager.RaiseAllocationFailure();
END_IF

_Workflow.RegisterChild(child := tryCatchAct^);
_ThrowingActivity.ShouldThrow := TRUE;

catchAct := __NEW(RecoveryCatchTestActivity(workflow := _Workflow));

IF catchAct = 0 THEN
	TOF_Core.DynamicMemoryManager.RaiseAllocationFailure();
END_IF

_Workflow.RegisterChild(child := catchAct^);

tryCatchAct^.Configure(tryActivity := _ThrowingActivity, catchActivity := catchAct^);
whileBody^.AddChildActivity(activity := tryCatchAct^);

// Set root activity on workflow
_Workflow.SetRootActivity(rootActivity := rootSequence^);
END_METHOD

(*!
<summary>Checks all relational operators on homogeneous INT workflow values.</summary>
<description>
Installs a root to register ProducedCount and BatchTarget in the workflow scope before comparison.
Exercises reference-value and variable-to-variable configuration. The persistent condition owns its value snapshot.
</description>
<param name="assertions">Valid assertion context borrowed from the active case.</param>
*)
METHOD PRIVATE testCompareVariableCondition
VAR_INPUT
	assertions : REFERENCE TO TOF_Testing.Assertions;
END_VAR
VAR
	threshold10 : INT := 10;
	threshold5 : INT := 5;
END_VAR
VAR_INST
	//! <summary>Root activity kept alive for the lifetime of the comparison fixture.</summary>
	comparisonRoot : TOF_Workflow.DelayActivity(workflow := _Workflow);
END_VAR
_Workflow.SetRootActivity(rootActivity := comparisonRoot);
_Workflow.ProducedCount := 5;

// Literal comparisons
_ComparisonCondition.Configure(
	firstVariableName := 'ProducedCount',
	comparisonOperator := TOF_Workflow.COMPARISON_OPERATOR.LESS_THAN,
	referenceValue := threshold10
);
assertions.ThatBool(
	actual := _ComparisonCondition.Evaluate(activity := 0),
	message := "5 < 10 must be TRUE"
).IsTrue();

_ComparisonCondition.Configure(
	firstVariableName := 'ProducedCount',
	comparisonOperator := TOF_Workflow.COMPARISON_OPERATOR.GREATER_THAN,
	referenceValue := threshold10
);
assertions.ThatBool(
	actual := _ComparisonCondition.Evaluate(activity := 0),
	message := "5 > 10 must be FALSE"
).IsFalse();

_ComparisonCondition.Configure(
	firstVariableName := 'ProducedCount',
	comparisonOperator := TOF_Workflow.COMPARISON_OPERATOR.EQUAL,
	referenceValue := threshold5
);
assertions.ThatBool(
	actual := _ComparisonCondition.Evaluate(activity := 0),
	message := "5 == 5 must be TRUE"
).IsTrue();

_ComparisonCondition.Configure(
	firstVariableName := 'ProducedCount',
	comparisonOperator := TOF_Workflow.COMPARISON_OPERATOR.NOT_EQUAL,
	referenceValue := threshold5
);
assertions.ThatBool(
	actual := _ComparisonCondition.Evaluate(activity := 0),
	message := "5 != 5 must be FALSE"
).IsFalse();

_ComparisonCondition.Configure(
	firstVariableName := 'ProducedCount',
	comparisonOperator := TOF_Workflow.COMPARISON_OPERATOR.GREATER_THAN_OR_EQUAL,
	referenceValue := threshold5
);
assertions.ThatBool(
	actual := _ComparisonCondition.Evaluate(activity := 0),
	message := "5 >= 5 must be TRUE"
).IsTrue();

_ComparisonCondition.Configure(
	firstVariableName := 'ProducedCount',
	comparisonOperator := TOF_Workflow.COMPARISON_OPERATOR.LESS_THAN_OR_EQUAL,
	referenceValue := threshold10
);
assertions.ThatBool(
	actual := _ComparisonCondition.Evaluate(activity := 0),
	message := "5 <= 10 must be TRUE"
).IsTrue();

// Variable-to-variable comparisons
_Workflow.BatchTarget := 10;
_ComparisonCondition.ConfigureVariable(
	firstVariableName := 'ProducedCount',
	comparisonOperator := TOF_Workflow.COMPARISON_OPERATOR.LESS_THAN,
	secondVariableName := 'BatchTarget'
);
assertions.ThatBool(
	actual := _ComparisonCondition.Evaluate(activity := 0),
	message := "ProducedCount (5) < BatchTarget (10) must be TRUE"
).IsTrue();

_ComparisonCondition.ConfigureVariable(
	firstVariableName := 'ProducedCount',
	comparisonOperator := TOF_Workflow.COMPARISON_OPERATOR.GREATER_THAN,
	secondVariableName := 'BatchTarget'
);
assertions.ThatBool(
	actual := _ComparisonCondition.Evaluate(activity := 0),
	message := "ProducedCount (5) > BatchTarget (10) must be FALSE"
).IsFalse();
END_METHOD

(*!
<summary>Checks numeric pair dispatch across widths, signedness and integer/floating-point representations.</summary>
<description>
Exercises both configuration paths and reversed operands, including an integer immediately above 2^53.
An explicit byte comparer must override automatic numeric ordering. Fixtures and copied references belong to
persistent suite fields; no resource-owning local function block relies on exception stack unwinding.
</description>
<param name="assertions">Valid assertion context borrowed from the active case.</param>
*)
METHOD PRIVATE testMixedNumericComparison
VAR_INPUT
	assertions : REFERENCE TO TOF_Testing.Assertions;
END_VAR
VAR
	customResult : BOOL;
END_VAR
_PairComparisonCondition.Comparer := 0;
_PairComparisonCondition.BindPlcVariable(name := 'NumericNarrow', plcVariable := _ComparisonNarrowInteger);
_PairComparisonCondition.BindPlcVariable(name := 'NumericWide', plcVariable := _ComparisonWideInteger);
_PairComparisonCondition.BindPlcVariable(name := 'NumericSigned', plcVariable := _ComparisonSignedInteger);
_PairComparisonCondition.BindPlcVariable(name := 'NumericUnsigned', plcVariable := _ComparisonUnsignedInteger);
_PairComparisonCondition.BindPlcVariable(name := 'NumericFloat', plcVariable := _ComparisonFloatingValue);

_PairComparisonCondition.ConfigureVariable(
	firstVariableName := 'NumericWide',
	comparisonOperator := TOF_Workflow.COMPARISON_OPERATOR.GREATER_THAN,
	secondVariableName := 'NumericNarrow'
);
assertions.ThatBool(
	actual := _PairComparisonCondition.Evaluate(activity := 0),
	message := "LINT 128 must exceed SINT 127"
).IsTrue();

_PairComparisonCondition.ConfigureVariable(
	firstVariableName := 'NumericNarrow',
	comparisonOperator := TOF_Workflow.COMPARISON_OPERATOR.LESS_THAN,
	secondVariableName := 'NumericWide'
);
assertions.ThatBool(
	actual := _PairComparisonCondition.Evaluate(activity := 0),
	message := "SINT 127 must precede LINT 128"
).IsTrue();

_PairComparisonCondition.Configure(
	firstVariableName := 'NumericWide',
	comparisonOperator := TOF_Workflow.COMPARISON_OPERATOR.GREATER_THAN,
	referenceValue := _ComparisonNarrowInteger
);
assertions.ThatBool(
	actual := _PairComparisonCondition.Evaluate(activity := 0),
	message := "A narrow reference must retain its value"
).IsTrue();

_PairComparisonCondition.Configure(
	firstVariableName := 'NumericNarrow',
	comparisonOperator := TOF_Workflow.COMPARISON_OPERATOR.LESS_THAN,
	referenceValue := _ComparisonWideInteger
);
assertions.ThatBool(
	actual := _PairComparisonCondition.Evaluate(activity := 0),
	message := "A wide reference must retain its value"
).IsTrue();

_PairComparisonCondition.ConfigureVariable(
	firstVariableName := 'NumericSigned',
	comparisonOperator := TOF_Workflow.COMPARISON_OPERATOR.LESS_THAN,
	secondVariableName := 'NumericUnsigned'
);
assertions.ThatBool(
	actual := _PairComparisonCondition.Evaluate(activity := 0),
	message := "INT -1 must precede UINT maximum"
).IsTrue();

_PairComparisonCondition.ConfigureVariable(
	firstVariableName := 'NumericUnsigned',
	comparisonOperator := TOF_Workflow.COMPARISON_OPERATOR.GREATER_THAN,
	secondVariableName := 'NumericSigned'
);
assertions.ThatBool(
	actual := _PairComparisonCondition.Evaluate(activity := 0),
	message := "UINT maximum must exceed INT -1"
).IsTrue();

_PairComparisonCondition.Configure(
	firstVariableName := 'NumericSigned',
	comparisonOperator := TOF_Workflow.COMPARISON_OPERATOR.LESS_THAN,
	referenceValue := _ComparisonUnsignedInteger
);
assertions.ThatBool(
	actual := _PairComparisonCondition.Evaluate(activity := 0),
	message := "A copied UINT reference must not be read as signed INT"
).IsTrue();

_PairComparisonCondition.Configure(
	firstVariableName := 'NumericUnsigned',
	comparisonOperator := TOF_Workflow.COMPARISON_OPERATOR.GREATER_THAN,
	referenceValue := _ComparisonSignedInteger
);
assertions.ThatBool(
	actual := _PairComparisonCondition.Evaluate(activity := 0),
	message := "A copied negative INT reference must remain negative"
).IsTrue();

// Adjacent integers above the exact binary64 integer range must not be rounded to equality.
_ComparisonWideInteger := LINT#9007199254740993;
_ComparisonFloatingValue := LREAL#9007199254740992.0;

_PairComparisonCondition.ConfigureVariable(
	firstVariableName := 'NumericWide',
	comparisonOperator := TOF_Workflow.COMPARISON_OPERATOR.GREATER_THAN,
	secondVariableName := 'NumericFloat'
);
assertions.ThatBool(
	actual := _PairComparisonCondition.Evaluate(activity := 0),
	message := "Mixed ordering must preserve 2^53 + 1"
).IsTrue();

_PairComparisonCondition.ConfigureVariable(
	firstVariableName := 'NumericFloat',
	comparisonOperator := TOF_Workflow.COMPARISON_OPERATOR.LESS_THAN,
	secondVariableName := 'NumericWide'
);
assertions.ThatBool(
	actual := _PairComparisonCondition.Evaluate(activity := 0),
	message := "Reversed mixed ordering must remain exact"
).IsTrue();

_PairComparisonCondition.Configure(
	firstVariableName := 'NumericWide',
	comparisonOperator := TOF_Workflow.COMPARISON_OPERATOR.GREATER_THAN,
	referenceValue := _ComparisonFloatingValue
);
assertions.ThatBool(
	actual := _PairComparisonCondition.Evaluate(activity := 0),
	message := "A copied floating reference must compare exactly"
).IsTrue();

_PairComparisonCondition.ConfigureVariable(
	firstVariableName := 'NumericSigned',
	comparisonOperator := TOF_Workflow.COMPARISON_OPERATOR.EQUAL,
	secondVariableName := 'NumericUnsigned'
);
_PairComparisonCondition.Comparer := TOF_Comparison.StandardComparers.ByteArrayComparer;
customResult := _PairComparisonCondition.Evaluate(activity := 0);
_PairComparisonCondition.Comparer := 0;

assertions.ThatBool(
	actual := customResult,
	message := "An explicit byte comparer must see identical signed and unsigned bytes"
).IsTrue();
assertions.ThatBool(
	actual := _PairComparisonCondition.Evaluate(activity := 0),
	message := "Automatic numeric equality must differ"
).IsFalse();
END_METHOD

